	IF NOT bBusy THEN
		fbRun_Color_RTRIG(CLK:=bSetColor, Q=> );
		IF fbRun_Color_RTRIG.Q THEN
			bRunColorWriteCycle:= TRUE;
		END_IF
	
		fbCycleReadTC_TON(IN:= bReadActualTC , PT:=T#1S , Q=> , ET=> );
	
		IF NOT bInitColor AND fActualTcColor = 0 THEN
			bRunColorWriteCycle:=TRUE;
		END_IF

	//Check for correct color in ballast 
	fbColorCheck(IN:= NOT fbColorCheck.Q , PT:= T#2S, Q=> , ET=> );	
	IF fbColorCheck.Q THEN
		IF fColourTemperatureTc <> fActualTcColor  THEN
			bRunColorWriteCycle:=TRUE;			
		END_IF
	END_IF

	
		IF  bRunColorWriteCycle AND NOT GVL_DALI.arrbBlockDTR[nDaliLine] THEN
			bBusy:= TRUE;
			A_ResetRoutine();
			nStep:= 10;
			nErrorID:= 0;
			iStepBeforeError:= 0;	
			GVL_DALI.arrbBlockDTR[nDaliLine] := TRUE;
		END_IF
		
		IF fbCycleReadTC_TON.Q THEN
			bBusy:= TRUE;
			bReadTC:= FALSE;
			A_ResetRoutine();
			nStep:= 100;
			nErrorID:= 0;
			iStepBeforeError:= 0;
		END_IF
	END_IF
	
(* - - - - - - - - - - - - - - - - - - - - - - - - *)
10:(*Set color temperatur to ballast*)
	bStart:= TRUE;
	A_DALICmdSetColourTemperatureTc();
	IF NOT bActionBusy	THEN
		IF bError	THEN
			GVL_DALI.arrbBlockDTR[nDaliLine]:= FALSE;
			nStep:= 0;
		ELSE
			bStart := FALSE;
			nStep:= 11;
		END_IF
	END_IF

11: (* Activate the color temp in ballast*)

	A_DALICmdActivate_DT8();
	
	IF NOT bActionBusy	THEN
		IF bError	THEN
			GVL_DALI.arrbBlockDTR[nDaliLine]:= FALSE;
			nStep:= 0;
		ELSE
			bStart := FALSE;
			nStep:= 100;	
		END_IF
	END_IF	

100: (*Read back current color*)

	A_DALIQueryColourTc();
	IF NOT bActionBusy	THEN
		nStep:= 101;
	END_IF

101: (*Read back color Status*)

	A_DALIQueryColourStatus();
	IF NOT bActionBusy	THEN
		nStep:= 888;
	END_IF
		
888: (*Done step*)
	bBusy:= FALSE;
	nStep:=0;
	nErrorID:= 0;
	iStepBeforeError:= 0;
	bRunColorWriteCycle:= FALSE;
	bInitColor:= TRUE;
	GVL_DALI.arrbBlockDTR[nDaliLine]:= FALSE;
ELSE
	nStep := 0;
END_CASE

//Checking if this FB blocks DT_Telegrams for other ballast

fbDTBlockTimer(IN:=GVL_DALI.arrbBlockDTR[nDaliLine] AND (nStep > 0) AND NOT fbDTBlockTimer.Q , PT:= T#20S , Q=> , ET=> );

IF fbDTBlockTimer.Q THEN
	nStep := 0;
	GVL_DALI.arrbBlockDTR[nDaliLine]:= FALSE;
END_IF

	fActualTcColor := MIREK_TO_KELVIN(fbDALI209QueryColourTc.nColourValue) ;
	nActualColorStatus := fbDALI209QueryColourStatus.nColourStatus;

ACTION A_DALICmdActivate_DT8:
IF eAddressType= E_DALIAddressType.Group THEN
	byAddr		:= byGrpAdr;
	eAddrType	:= E_DALIAddressType.Group;
END_IF

IF eAddressType= E_DALIAddressType.Short THEN
	byAddr		:= byShrtAdr;
	eAddrType	:= E_DALIAddressType.Short;
END_IF

	bActionBusy	:= TRUE;

	fbDALI209Activate(
		bError=> , 
		ipResultMessage=> , 
		bStart:= TRUE, 
		nAddress:= byAddr , 
		eAddressType:= eAddressType, 
		eCommandPriority:=eCommandPriority ,
		bBusy=> );
	

	IF (NOT fbDALI209Activate.bBusy) THEN
		IF fbDALI209Activate.bError THEN
			bError := TRUE;
			nErrorId := fbDALI209Activate.ipResultMessage.nEventId;
		END_IF
		bActionBusy		:= FALSE;
		fbDALI209Activate(bStart:= FALSE);
	END_IF
END_ACTION

ACTION A_DALICmdSetColourTemperatureTc:
IF eAddressType= E_DALIAddressType.Group THEN
	byAddr		:= byGrpAdr;
	eAddrType	:= E_DALIAddressType.Group;
END_IF

IF eAddressType= E_DALIAddressType.Short THEN
	byAddr		:= byShrtAdr;
	eAddrType	:= E_DALIAddressType.Short;
END_IF

	bActionBusy	:= TRUE;

	fbDALI209SetColourTemperatureTc(
		bError=> , 
		ipResultMessage=> , 
		bStart:= TRUE, 
		nAddress:= byAddr , 
		eAddressType:= eAddressType, 
		eCommandPriority:=eCommandPriority , 
		bBusy=> , 
		nColourTemperatureTc:= KELVIN_TO_MIREK(fColourTemperatureTc)
	);
	
	
	
	IF (NOT fbDALI209SetColourTemperatureTc.bBusy) THEN
		IF fbDALI209SetColourTemperatureTc.bError THEN
			bError := TRUE;
			nErrorId := fbDALI209SetColourTemperatureTc.ipResultMessage.nEventId;
		END_IF
		bActionBusy		:= FALSE;
		fbDALI209SetColourTemperatureTc(bStart:= FALSE);
	END_IF
END_ACTION

ACTION A_DALIQueryColourStatus:

	byAddr:= byShrtAdr;

	bActionBusy	:= TRUE;


	fbDALI209QueryColourStatus(
		bError=> , 
		ipResultMessage=> , 
		bStart:= TRUE , 
		nAddress:=byAddr , 
		eAddressType:= Tc3_DALI.E_DALIAddressType.Short, 
		eCommandPriority:= Tc3_DALI.E_DALICommandPriority.Low, 
		bBusy=> , 
		nColourStatus=> );	
	

	IF (NOT fbDALI209QueryColourStatus.bBusy) THEN
		IF fbDALI209QueryColourStatus.bError THEN
			bError := TRUE;
			nErrorId := fbDALI209QueryColourStatus.ipResultMessage.nEventId;
		END_IF
		bActionBusy		:= FALSE;
		fbDALI209QueryColourStatus(bStart:= FALSE);
	END_IF
END_ACTION

ACTION A_DALIQueryColourTc:

	byAddr:= byShrtAdr;

	bActionBusy	:= TRUE;


	fbDALI209QueryColourTc(
		bError=> , 
		ipResultMessage=> , 
		bStart:= TRUE , 
		nAddress:=byAddr , 
		eAddressType:= Tc3_DALI.E_DALIAddressType.Short, 
		eCommandPriority:= Tc3_DALI.E_DALICommandPriority.Low, 
		bBusy=> , 
		eColourValue:= Tc3_DALI.E_DALIColourValue.ColourTemperatureTc , 
		nColourValue=> );	
	

	IF (NOT fbDALI209QueryColourTc.bBusy) THEN
		IF fbDALI209QueryColourTc.bError THEN
			bError := TRUE;
			nErrorId := fbDALI209QueryColourTc.ipResultMessage.nEventId;
		END_IF
		bActionBusy		:= FALSE;
		fbDALI209QueryColourTc(bStart:= FALSE);
	END_IF
END_ACTION

ACTION A_ResetRoutine:

	bError     	:= FALSE;
	nErrorId	:= 0;

	fbDALI209SetColourTemperatureTc (bStart:= FALSE);
	fbDALI209QueryColourStatus(bStart:= FALSE);
	fbDALI209QueryColourTc(bStart:= FALSE);
	fbDALI209Activate(bStart:= FALSE);
END_ACTION

{attribute 'monitoring' := 'call'}
PROPERTY ipDALICommunication : Tc3_DALI.I_DALICommunication
GET
ipDALICommunication := THIS^.ipCommunication;
END_GET
SET
THIS^.ipCommunicationPreset := ipDALICommunication;
END_SET
END_PROPERTY

//| Apply the perset value of IpCommunication if available
//| Return codes:
//|   FALSE: no peset value available
//|   TRUE: has taken the preset value
{attribute 'hide'}
METHOD PRIVATE TrySetCommunication : BOOL
VAR_INPUT
END_VAR
IF ((THIS^.ipCommunication <> THIS^.ipCommunicationPreset) AND (THIS^.ipCommunicationPreset <> 0)) THEN
	THIS^.ipCommunication := THIS^.ipCommunicationPreset;
	THIS^.fbDALI209Activate.ipDALICommunication := THIS^.ipCommunication;
	THIS^.fbDALI209SetColourTemperatureTc.ipDALICommunication := THIS^.ipCommunication;
	THIS^.fbDALI209QueryColourStatus.ipDALICommunication := THIS^.ipCommunication;
	THIS^.fbDALI209QueryColourTc.ipDALICommunication := THIS^.ipCommunication;
	TrySetCommunication := TRUE;
ELSE
	TrySetCommunication := FALSE;
END_IF
END_METHOD

END_FUNCTION_BLOCK

// POUs/DALI/DALI_Devices/BEG/FB_BEG_PD2N_1Pcs
FUNCTION_BLOCK FB_BEG_PD2N_1Pcs
VAR_INPUT
	byShrtAdr					: BYTE;
	bInitialize					: BOOL := TRUE;
	ipCommunication				: I_DALICommunication;
	DALI_LINE_NUM				: INT := 1;	
END_VAR
VAR_OUTPUT
	bInitErr: BOOL;
	bInitDone: BOOL;
END_VAR
VAR
	fbBEGPD2N					: FB_DALI_BEG_PD2N_BMS_V8_FC(0);
	
	fbDelaySetupDALIDevice		: TON;
	tDelayTime					: TIME;
	bInitSensor					: BOOL;
	fbInitDone					: F_TRIG;
	bInitializing				: BOOL;

	bQueryOccupancy				: BOOL;
	bQueryBrightness			: BOOL;

	eEventPriorityOccupancy		: E_DALIEventPriority := E_DALIEVENTPRIORITY.Middle;
	nHoldTimerOccupancy			: WORD := 5; // Value in s. 	
	nReportTimerOccupancy		: BYTE := 120; // Value in s, Preset manufacturer value
	nDeadtimeTimerOccupancy		: WORD := 100; // Value in ms, Predefined Value of DALI Standard
	bCancelHoldTimerOccupancy	: BOOL;
	nSensitivityOccupancy		: BYTE:= 3; //setting Sensivity (0..4) 0 (Off), 1 (Min), 2(Low), 3(High) and 4 (Max)

	bEnableLuxEvent				: BOOL;
	eEventPriorityBrightness	: E_DALIEventPriority := E_DALIEVENTPRIORITY.Middle;
	nDeadtimeTimerBrightness	: WORD := 1500; // Value in ms, Predefined Value of DALI Standard
	nHysteresisBrightness		: BYTE := 2; // Value in %
	nHysteresisMinBrightness	: BYTE := 10; // Absolute Value, depending on the manufacturer specific resolution
	nReportTimerBrightness		: BYTE := 120; // Value in s, Preset manufacturer value

	bAutoRead					: BOOL;
	fbAutoRequestBrightness_TON	: TOF;
	bInitTimeOut: BOOL;
	fbInitTimeOut: Ton;
	nCheckIdx: INT;
	bInitScalesDone: BOOL;
END_VAR
VAR_IN_OUT
	stPirSensorData				: ST_DALI_Sensor;
	arrSensorScales				: ARRAY [1.. 10] OF ST_DALI_SensorScaleMode;
END_VAR

fbBEGPD2N.ipDALICommunication := ipCommunication;

IF NOT bInitScalesDone THEN
	FOR nCheckIdx:= 1 TO 10 DO
		IF arrSensorScales[nCheckIdx].fMeassureMaxSensor = 0 THEN
			arrSensorScales[nCheckIdx].fMeassureMaxSensor := 1;
		END_IF
		IF arrSensorScales[nCheckIdx].fReadMaxSensor = 0 THEN
			arrSensorScales[nCheckIdx].fReadMaxSensor := 1;
		END_IF
	END_FOR
	bInitScalesDone := TRUE;
END_IF

IF ipCommunication <> 0 THEN
	A_BEG_PD2N_1();
END_IF

ACTION A_BEG_PD2N_1:
//Setup parameters
	//Setup Motion part of sensor (Instance 0)
	fbBEGPD2N.bEnableOccupancy := TRUE ;
	fbBEGPD2N.eEventPriorityOccupancy:= eEventPriorityOccupancy;
	fbBEGPD2N.nHoldTimerOccupancy := nHoldTimerOccupancy ;
	fbBEGPD2N.nReportTimerOccupancy := nReportTimerOccupancy;
	fbBEGPD2N.nDeadtimeTimerOccupancy:= nDeadtimeTimerOccupancy;
	fbBEGPD2N.nSensitivityOccupancy:= nSensitivityOccupancy;	
	
	//Setup Brightness part of sensor (Instance 1)
	fbBEGPD2N.bEnableBrightness := bEnableLuxEvent;
	fbBEGPD2N.eEventPriorityBrightness:= eEventPriorityBrightness;
	fbBEGPD2N.nDeadtimeTimerBrightness:= nDeadtimeTimerBrightness;
	fbBEGPD2N.nHysteresisBrightness:= nHysteresisBrightness;
	fbBEGPD2N.nHysteresisMinBrightness:= nHysteresisMinBrightness;
	fbBEGPD2N.nReportTimerBrightness:= nReportTimerBrightness;
	
	
	
//Calculate delay time for init sensor
tDelayTime := INT_TO_TIME((BYTE_TO_INT(byShrtAdr) * 400));	
fbDelaySetupDALIDevice(IN:= bInitialize AND NOT bInitDone , PT:=tDelayTime , Q=> , ET=> );	
	
IF fbDelaySetupDALIDevice.q AND NOT GVL_DALI.arrbBlockDTR[DALI_LINE_NUM] AND NOT bInitErr THEN
	bInitDone := FALSE;
	bInitErr := FALSE;
	bInitSensor:= TRUE;
	GVL_DALI.arrbBlockDTR[DALI_LINE_NUM]:= TRUE;
END_IF

fbAutoRequestBrightness_TON(IN:= NOT fbAutoRequestBrightness_TON.Q  AND NOT stPirSensorData.bQueryBrightness , PT:= (tDelayTime + T#10M) , Q=>bAutoRead , ET=> );

bQueryBrightness:= stPirSensorData.bQueryBrightness OR NOT bAutoRead;

fbBEGPD2N(
	bError=> , 
	ipResultMessage=> , 
	bInitialize:=  bInitSensor, 
	nShortAddress:= byShrtAdr, 
	nOptions:= , 
	bQueryOccupancy:= bQueryOccupancy, 
	bQueryBrightness:= bQueryBrightness, 
	bCancelHoldTimerOccupancy:= bCancelHoldTimerOccupancy, 
	bInitializing=> bInitializing , 
	bReadingOccupancy=> , 
	bReadingBrightness=> , 
	bOccupied=> stPirSensorData.bPrc, 
	nBrightnessLevel=> );


fbInitDone(CLK:=bInitSensor AND bInitializing );	
	IF fbInitDone.Q THEN
		IF NOT bInitTimeOut THEN
			bInitDone := TRUE;
			bInitErr := FALSE;
			GVL_DALI.arrbBlockDTR[DALI_LINE_NUM]:= FALSE;
		ELSE
			bInitErr := TRUE;
			GVL_DALI.arrbBlockDTR[DALI_LINE_NUM]:= FALSE;
		END_IF
	END_IF


fbInitTimeOut(IN:=bInitializing, PT:= T#10S); 

IF fbInitTimeOut.Q THEN
	bInitErr := TRUE;
	GVL_DALI.arrbBlockDTR[DALI_LINE_NUM]:= FALSE;
END_IF

stPirSensorData.bBrightnessRead:= fbBEGPD2N.bReadingBrightness ;

stPirSensorData.fBrightness:= F_fScale(0, arrSensorScales[1].fReadMaxSensor, 0, arrSensorScales[1].fMeassureMaxSensor, 0 , fbBEGPD2N.nBrightnessLevel);
END_ACTION

END_FUNCTION_BLOCK

// POUs/DALI/FUNs/F_fScale
FUNCTION F_fScale : REAL
VAR_INPUT
	fX0, fX1, fY0, fY1, fOffset : REAL;
	nRawValue	:UINT;
END_VAR
VAR
	fDeltaY: REAL;
	fDeltaX: REAL;

END_VAR
VAR_OUTPUT
END_VAR

fDeltaY:= fY1-fY0;
fDeltaX :=fX1-fX0;

IF fDeltaX <=0 THEN
	fDeltaX:=1;
END_IF

F_fScale:= (fDeltaY / fDeltaX) * UINT_TO_REAL(nRawValue) + fOffset;

END_FUNCTION

// POUs/DALI/DALI_Devices/ESYLux/Flat/FB_DALI_ESYLuxFlat_1Pcs
FUNCTION_BLOCK FB_DALI_ESYLuxFlat_1Pcs
VAR_INPUT
	byShrtAdr					: BYTE;
	bInitialize					: BOOL := TRUE;
	ipCommunication				: I_DALICommunication;
	DALI_LINE_NUM				: INT := 1;	
END_VAR
VAR_OUTPUT
END_VAR
VAR
	fbESYLux 					: FB_DALI_Esylux_PD_FLAT_360_BMS(0);
	
	fbDelaySetupDALIDevice		: TON;
	tDelayTime					: TIME;
	bInitSensor					: BOOL;
	fbInitDone					: F_TRIG;

	bQueryOccupancy				: BOOL;
	bQueryBrightness			: BOOL;

	bInitializing				: BOOL;

	eEventPriorityOccupancy		: E_DALIEventPriority := E_DALIEVENTPRIORITY.Middle;
	nHoldTimerOccupancy			: UINT := 5;
	nReportTimerOccupancy		: BYTE := 120; // Value in s, Preset manufacturer value
	nDeadtimeTimerOccupancy		: WORD := 100; // Value in ms, Predefined Value of DALI Standard
	bCancelHoldTimerOccupancy	: BOOL;
	nSensitivityOccupancy		: BYTE := 95; //setting Sensivity 0 = Low 100 = Max
	
	bEnableBrightness			: BOOL := FALSE;
	eEventPriorityBrightness	: E_DALIEventPriority := E_DALIEVENTPRIORITY.MiddleLow;
	nDeadtimeTimerBrightness	: WORD := 1500; // Value in ms, Predefined Value of DALI Standard
	nHysteresisBrightness		: BYTE := 5; // Value in %
	nHysteresisMinBrightness	: BYTE := 40; // Absolute Value, depending on the manufacturer specific resolution
	nReportTimerBrightness		: BYTE := 30; // Value in s, Preset manufacturer value

	bModeLED					: BOOL := FALSE; //LED mode: FALSE: LED disabled, TRUE: LED enabled
	nBrightnessLED				: USINT := 50; //LED brightness (5...100 %).
	
	bAutoRead					: BOOL;
	fbAutoRequestBrightness_TON	: TOF;
	bInitScalesDone				: BOOL;
	nCheckIdx					: INT;
	bInitDone					: BOOL;
	bInitErr					: BOOL;
	bInitTimeOut				: BOOL;
	fbInitTimeOut				: TON;
END_VAR
VAR_IN_OUT
	stPirSensorData				: ST_DALI_Sensor;
	arrSensorScales				: ARRAY [1.. 10] OF ST_DALI_SensorScaleMode;
END_VAR

fbESYLux.ipDALICommunication:= ipCommunication;

IF NOT bInitScalesDone THEN
	FOR nCheckIdx:= 1 TO 10 DO
		IF arrSensorScales[nCheckIdx].fMeassureMaxSensor = 0 THEN
			arrSensorScales[nCheckIdx].fMeassureMaxSensor := 1;
		END_IF
		IF arrSensorScales[nCheckIdx].fReadMaxSensor = 0 THEN
			arrSensorScales[nCheckIdx].fReadMaxSensor := 1;
		END_IF
	END_FOR
	bInitScalesDone := TRUE;
END_IF

IF ipCommunication <> 0 THEN
	A_ESYLux_1();
END_IF

ACTION A_ESYLux_1:
//Setup parameters
	//Setup Motion part of sensor (Instance 1)

	fbESYLux.bEnableOccupancy := TRUE;
	fbESYLux.eEventPriorityOccupancy:= eEventPriorityOccupancy;
	fbESYLux.nHoldTimerOccupancy := nHoldTimerOccupancy ;
	fbESYLux.nReportTimerOccupancy := nReportTimerOccupancy;
	fbESYLux.nDeadtimeTimerOccupancy:= nDeadtimeTimerOccupancy;
	fbESYLux.nSensitivityOccupancy:= nSensitivityOccupancy;
	
	
	//Setup Brightness part of sensor (Instance 2)
	fbESYLux.bEnableBrightness:= bEnableBrightness;
	fbESYLux.eEventPriorityBrightness:= eEventPriorityBrightness;
	fbESYLux.nDeadtimeTimerBrightness:= nDeadtimeTimerBrightness;
	fbESYLux.nHysteresisBrightness:= nHysteresisBrightness;
	fbESYLux.nHysteresisMinBrightness:= nHysteresisMinBrightness;
	fbESYLux.nReportTimerBrightness:= nReportTimerBrightness;

	fbESYLux.bModeLED:= bModeLED;
	fbESYLux.nBrightnessLED:= nBrightnessLED;
	
	
//Calculate delay time for init sensor
tDelayTime := INT_TO_TIME((BYTE_TO_INT(byShrtAdr) * 400));	
fbDelaySetupDALIDevice(IN:= bInitialize AND NOT bInitDone , PT:=tDelayTime , Q=> , ET=> );	
	
IF fbDelaySetupDALIDevice.q AND NOT GVL_DALI.arrbBlockDTR[DALI_LINE_NUM] AND NOT bInitErr THEN
	bInitDone := FALSE;
	bInitErr := FALSE;
	bInitSensor:= TRUE;
	GVL_DALI.arrbBlockDTR[DALI_LINE_NUM]:= TRUE;
END_IF

fbAutoRequestBrightness_TON(IN:= NOT fbAutoRequestBrightness_TON.Q  AND NOT stPirSensorData.bQueryBrightness , PT:= (tDelayTime + T#12M) , Q=>bAutoRead , ET=> );

bQueryBrightness:= stPirSensorData.bQueryBrightness OR NOT bAutoRead;

fbESYLux(
	bInitialize:= bInitSensor, 
	nShortAddress:= byShrtAdr, 
	nOptions:= , 
	bQueryPushButton:= , 
	bQueryOccupancy:= bQueryOccupancy, 
	bQueryBrightness:= bQueryBrightness, 
	bCancelHoldTimerOccupancy:= bCancelHoldTimerOccupancy, 
	bInitializing=> bInitializing , 
	bReadingPushButton=> , 
	bReadingOccupancy=> , 
	bReadingBrightness=> , 
	nPushButtonEvent=> , 
	bOccupied=> stPirSensorData.bPrc, 
	nBrightnessLevel=> );

fbInitDone(CLK:=bInitSensor AND bInitializing );	
	IF fbInitDone.Q THEN
		IF NOT bInitTimeOut THEN
			bInitDone := TRUE;
			bInitErr := FALSE;
			GVL_DALI.arrbBlockDTR[DALI_LINE_NUM]:= FALSE;
		ELSE
			bInitErr := TRUE;
			GVL_DALI.arrbBlockDTR[DALI_LINE_NUM]:= FALSE;
		END_IF
	END_IF


fbInitTimeOut(IN:=bInitializing, PT:= T#10S); 

IF fbInitTimeOut.Q THEN
	bInitErr := TRUE;
	GVL_DALI.arrbBlockDTR[DALI_LINE_NUM]:= FALSE;
END_IF

stPirSensorData.bBrightnessRead:= fbESYLux.bReadingBrightness ;

stPirSensorData.fBrightness:= F_fScale(0, arrSensorScales[1].fReadMaxSensor, 0, arrSensorScales[1].fMeassureMaxSensor, 0 , fbESYLux.nBrightnessLevel);
END_ACTION

END_FUNCTION_BLOCK

// POUs/DALI/DALI_Devices/ESYLux/FB_DALI_ESYLux_1Pcs
FUNCTION_BLOCK FB_DALI_ESYLux_1Pcs
VAR_INPUT
	byShrtAdr					: BYTE;
	bInitialize					: BOOL := TRUE;
	ipCommunication				: I_DALICommunication;
	DALI_LINE_NUM				: INT := 1;	
END_VAR
VAR_OUTPUT
END_VAR
VAR
	fbESYLux 					: FB_DALI_Esylux_PD_C_360_BMS(0);
	
	fbDelaySetupDALIDevice		: TON;
	tDelayTime					: TIME;
	bInitSensor					: BOOL;
	fbInitDone					: F_TRIG;

	bQueryOccupancy				: BOOL;
	bQueryBrightness			: BOOL;

	bInitializing				: BOOL;

	eEventPriorityOccupancy		: E_DALIEventPriority := E_DALIEVENTPRIORITY.Middle;
	nHoldTimerOccupancy			: UINT := 5;
	nReportTimerOccupancy		: BYTE := 120; // Value in s, Preset manufacturer value
	nDeadtimeTimerOccupancy		: WORD := 100; // Value in ms, Predefined Value of DALI Standard
	bCancelHoldTimerOccupancy	: BOOL;
	nSensitivityOccupancy		: BYTE := 95; //setting Sensivity 0 = Low 100 = Max
	
	bEnableBrightness			: BOOL := FALSE;
	eEventPriorityBrightness	: E_DALIEventPriority := E_DALIEVENTPRIORITY.MiddleLow;
	nDeadtimeTimerBrightness	: WORD := 1500; // Value in ms, Predefined Value of DALI Standard
	nHysteresisBrightness		: BYTE := 5; // Value in %
	nHysteresisMinBrightness	: BYTE := 40; // Absolute Value, depending on the manufacturer specific resolution
	nReportTimerBrightness		: BYTE := 30; // Value in s, Preset manufacturer value

	bModeLED					: BOOL := FALSE; //LED mode: FALSE: LED disabled, TRUE: LED enabled
	nBrightnessLED				: USINT := 50; //LED brightness (5...100 %).
	
	bAutoRead					: BOOL;
	fbAutoRequestBrightness_TON	: TOF;
	bInitScalesDone				: BOOL;
	nCheckIdx					: INT;
	bInitDone					: BOOL;
	bInitErr					: BOOL;
	bInitTimeOut				: BOOL;
	fbInitTimeOut				: TON;
END_VAR
VAR_IN_OUT
	stPirSensorData				: ST_DALI_Sensor;
	arrSensorScales				: ARRAY [1.. 10] OF ST_DALI_SensorScaleMode;
END_VAR

fbESYLux.ipDALICommunication:= ipCommunication;

IF NOT bInitScalesDone THEN
	FOR nCheckIdx:= 1 TO 10 DO
		IF arrSensorScales[nCheckIdx].fMeassureMaxSensor = 0 THEN
			arrSensorScales[nCheckIdx].fMeassureMaxSensor := 1;
		END_IF
		IF arrSensorScales[nCheckIdx].fReadMaxSensor = 0 THEN
			arrSensorScales[nCheckIdx].fReadMaxSensor := 1;
		END_IF
	END_FOR
	bInitScalesDone := TRUE;
END_IF

IF ipCommunication <> 0 THEN
	A_ESYLux_1();
END_IF

ACTION A_ESYLux_1:
//Setup parameters
	//Setup Motion part of sensor (Instance 0)

	fbESYLux.bEnableOccupancy := TRUE;
	fbESYLux.eEventPriorityOccupancy:= eEventPriorityOccupancy;
	fbESYLux.nHoldTimerOccupancy := nHoldTimerOccupancy ;
	fbESYLux.nReportTimerOccupancy := nReportTimerOccupancy;
	fbESYLux.nDeadtimeTimerOccupancy:= nDeadtimeTimerOccupancy;
	fbESYLux.nSensitivityOccupancy:= nSensitivityOccupancy;
	
	
	//Setup Brightness part of sensor (Instance 1)
	fbESYLux.bEnableBrightness:= bEnableBrightness;
	fbESYLux.eEventPriorityBrightness:= eEventPriorityBrightness;
	fbESYLux.nDeadtimeTimerBrightness:= nDeadtimeTimerBrightness;
	fbESYLux.nHysteresisBrightness:= nHysteresisBrightness;
	fbESYLux.nHysteresisMinBrightness:= nHysteresisMinBrightness;
	fbESYLux.nReportTimerBrightness:= nReportTimerBrightness;

	fbESYLux.bModeLED:= bModeLED;
	fbESYLux.nBrightnessLED:= nBrightnessLED;
	
	
//Calculate delay time for init sensor
tDelayTime := INT_TO_TIME((BYTE_TO_INT(byShrtAdr) * 400));	
fbDelaySetupDALIDevice(IN:= bInitialize AND NOT bInitDone , PT:=tDelayTime , Q=> , ET=> );	
	
IF fbDelaySetupDALIDevice.q AND NOT GVL_DALI.arrbBlockDTR[DALI_LINE_NUM] AND NOT bInitErr THEN
	bInitDone := FALSE;
	bInitErr := FALSE;
	bInitSensor:= TRUE;
	GVL_DALI.arrbBlockDTR[DALI_LINE_NUM]:= TRUE;
END_IF

fbAutoRequestBrightness_TON(IN:= NOT fbAutoRequestBrightness_TON.Q  AND NOT stPirSensorData.bQueryBrightness , PT:= (tDelayTime + T#12M) , Q=>bAutoRead , ET=> );

bQueryBrightness:= stPirSensorData.bQueryBrightness OR NOT bAutoRead;

fbESYLux(
	bInitialize:= bInitSensor, 
	nShortAddress:= byShrtAdr, 
	nOptions:= , 
	bQueryPushButton1:= , 
	bQueryPushButton2:= , 
	bQueryOccupancy:= bQueryOccupancy, 
	bQueryBrightness:= bQueryBrightness, 
	bCancelHoldTimerOccupancy:= bCancelHoldTimerOccupancy, 
	bInitializing=> bInitializing , 
	bReadingPushButton1=> , 
	bReadingPushButton2=> , 
	bReadingOccupancy=> , 
	bReadingBrightness=> , 
	nPushButton1Event=> , 
	nPushButton2Event=> , 
	bOccupied=> stPirSensorData.bPrc, 
	nBrightnessLevel=> );


fbInitDone(CLK:=bInitSensor AND bInitializing );	
	IF fbInitDone.Q THEN
		IF NOT bInitTimeOut THEN
			bInitDone := TRUE;
			bInitErr := FALSE;
			GVL_DALI.arrbBlockDTR[DALI_LINE_NUM]:= FALSE;
		ELSE
			bInitErr := TRUE;
			GVL_DALI.arrbBlockDTR[DALI_LINE_NUM]:= FALSE;
		END_IF
	END_IF


fbInitTimeOut(IN:=bInitializing, PT:= T#10S); 

IF fbInitTimeOut.Q THEN
	bInitErr := TRUE;
	GVL_DALI.arrbBlockDTR[DALI_LINE_NUM]:= FALSE;
END_IF

stPirSensorData.bBrightnessRead:= fbESYLux.bReadingBrightness ;

stPirSensorData.fBrightness:= F_fScale(0, arrSensorScales[1].fReadMaxSensor, 0, arrSensorScales[1].fMeassureMaxSensor, 0 , fbESYLux.nBrightnessLevel);
END_ACTION

END_FUNCTION_BLOCK

// POUs/DALI/DALI_Devices/ESYLux/FB_DALI_ESYLux_2Pcs
FUNCTION_BLOCK FB_DALI_ESYLux_2Pcs
VAR_INPUT
	byShrtAdr					: BYTE;
	bInitialize					: BOOL := TRUE;
	ipCommunication				: I_DALICommunication;
	DALI_LINE_NUM				: INT := 1;	
END_VAR
VAR_OUTPUT
	arrInitErr: ARRAY [1.. nNumberOfSensors] OF BOOL;
	arrInitDone: ARRAY [1.. nNumberOfSensors] OF BOOL;
END_VAR
VAR
	arrEsylux_PD_C				: ARRAY [1.. nNumberOfSensors] OF FB_DALI_Esylux_PD_C_360_BMS(0);
	
	arrDelaySetupDALIDevice		: ARRAY [1.. nNumberOfSensors] Of TON;
	arrtDelayTime				: ARRAY [1.. nNumberOfSensors] OF TIME;
	arrInitSensor				: ARRAY [1.. nNumberOfSensors] OF BOOL;
	arrInitDone_FTrig			: ARRAY [1.. nNumberOfSensors] OF F_TRIG;
	arrInitializing				: ARRAY [1.. nNumberOfSensors] OF BOOL;

	bQueryBrightness 			: BOOL;
	bQueryOccupancy				: BOOL;

	eEventPriorityOccupancy		: E_DALIEventPriority := E_DALIEVENTPRIORITY.Middle;
	nHoldTimerOccupancy			: UINT := 5;
	nReportTimerOccupancy		: BYTE := 120; // Value in s, Preset manufacturer value
	nDeadtimeTimerOccupancy		: WORD := 100; // Value in ms, Predefined Value of DALI Standard
	bCancelHoldTimerOccupancy	: BOOL;
	nSensitivityOccupancy		: BYTE := 95; //setting Sensivity 0 = Low 100 = Max
	
	bEnableBrightness			: BOOL := FALSE;
	eEventPriorityBrightness	: E_DALIEventPriority := E_DALIEVENTPRIORITY.MiddleLow;
	nDeadtimeTimerBrightness	: WORD := 1500; // Value in ms, Predefined Value of DALI Standard
	nHysteresisBrightness		: BYTE := 5; // Value in %
	nHysteresisMinBrightness	: BYTE := 40; // Absolute Value, depending on the manufacturer specific resolution
	nReportTimerBrightness		: BYTE := 30; // Value in s, Preset manufacturer value

	bModeLED					: BOOL := FALSE; //LED mode: FALSE: LED disabled, TRUE: LED enabled
	nBrightnessLED				: USINT := 50; //LED brightness (5...100 %).

	bAutoRead					: BOOL;
	fbAutoRequestBrightness_TON	: TOF;
	bInitTimeOut				: BOOL;
	fbInitTimeOut				: ARRAY [1.. nNumberOfSensors] OF TON;
	nIdxScan					: BYTE;
	nPirIdxOn					: BYTE;
	nBrightnessIdx				: BYTE;
	fBrightness_1				: REAL;
	fBrightness_2				: REAL;
	fBrightness_3				: REAL;
	bInitDone					: BOOL;
	bInitScalesDone				: BOOL;
	
	nCheckIdx: INT;
END_VAR
VAR_IN_OUT
	stPirSensorData				: ST_DALI_Sensor;
	arrSensorScales				: ARRAY [1.. 10] OF ST_DALI_SensorScaleMode;
END_VAR

VAR CONSTANT
	nNumberOfSensors: BYTE := 2;
END_VAR

arrEsylux_PD_C[1].ipDALICommunication := ipCommunication;
arrEsylux_PD_C[2].ipDALICommunication := ipCommunication;


IF NOT bInitScalesDone THEN
	FOR nCheckIdx:= 1 TO 10 DO
		IF arrSensorScales[nCheckIdx].fMeassureMaxSensor = 0 THEN
			arrSensorScales[nCheckIdx].fMeassureMaxSensor := 1;
		END_IF
		IF arrSensorScales[nCheckIdx].fReadMaxSensor = 0 THEN
			arrSensorScales[nCheckIdx].fReadMaxSensor := 1;
		END_IF
	END_FOR
	bInitScalesDone := TRUE;
END_IF

IF ipCommunication <> 0 THEN
	A_ESYLux_2Pcs();
END_IF

ACTION A_ESYLux_2Pcs:


FOR nIdxScan := 1 TO nNumberOfSensors DO
	//Setup parameters
	//Setup Motion part of sensor (Instance 0)
	arrEsylux_PD_C[nIdxScan].bEnableOccupancy := TRUE;
	arrEsylux_PD_C[nIdxScan].eEventPriorityOccupancy:= eEventPriorityOccupancy;
	arrEsylux_PD_C[nIdxScan].nHoldTimerOccupancy := nHoldTimerOccupancy ;
	arrEsylux_PD_C[nIdxScan].nDeadtimeTimerOccupancy:= 	nDeadtimeTimerOccupancy;
	arrEsylux_PD_C[nIdxScan].nReportTimerOccupancy:= nReportTimerOccupancy;
	arrEsylux_PD_C[nIdxScan].nSensitivityOccupancy:= 100;
	
	//Setup Brightness part of sensor (Instance 1)
	arrEsylux_PD_C[nIdxScan].bEnableBrightness:= bEnableBrightness;
	arrEsylux_PD_C[nIdxScan].eEventPriorityBrightness:= eEventPriorityBrightness;
	arrEsylux_PD_C[nIdxScan].nDeadtimeTimerBrightness:= nDeadtimeTimerBrightness;
	arrEsylux_PD_C[nIdxScan].nHysteresisBrightness:= nHysteresisBrightness;
	arrEsylux_PD_C[nIdxScan].nHysteresisMinBrightness:= nHysteresisMinBrightness;
	arrEsylux_PD_C[nIdxScan].nReportTimerBrightness:= nReportTimerBrightness;

	arrEsylux_PD_C[nIdxScan].bModeLED:= bModeLED;
	arrEsylux_PD_C[nIdxScan].nBrightnessLED:= nBrightnessLED;
	
		
		
	//Calculate delay time for init sensor
	arrtDelayTime[nIdxScan] := INT_TO_TIME((BYTE_TO_INT((byShrtAdr + nIdxScan)-1) * 400));	
	arrDelaySetupDALIDevice[nIdxScan](IN:= bInitialize , PT:=arrtDelayTime[nIdxScan] , Q=> , ET=> );	
		
	IF arrDelaySetupDALIDevice[nIdxScan].q AND NOT GVL_DALI.arrbBlockDTR[DALI_LINE_NUM] AND NOT (arrInitDone[nIdxScan] OR arrInitErr[nIdxScan]) THEN
		arrInitSensor[nIdxScan]:= TRUE;
		GVL_DALI.arrbBlockDTR[DALI_LINE_NUM]:= TRUE;
	END_IF
	
	bQueryBrightness:= stPirSensorData.bQueryBrightness OR NOT bAutoRead;
	
	fbAutoRequestBrightness_TON(IN:= NOT fbAutoRequestBrightness_TON.Q  AND NOT stPirSensorData.bQueryBrightness , PT:= (arrtDelayTime[nIdxScan] + T#12M) , Q=>bAutoRead , ET=> );
	
	bQueryOccupancy:= NOT bAutoRead OR stPirSensorData.bQueryBrightness;
	
	arrEsylux_PD_C[nIdxScan](
		bError=> , 
		ipResultMessage=> , 
		bInitialize:=  arrInitSensor[nIdxScan], 
		nShortAddress:= (byShrtAdr + nIdxScan)-1 , 
		nOptions:= , 
		bQueryOccupancy:= bQueryOccupancy, 
		bQueryBrightness:= bQueryBrightness, 
		bCancelHoldTimerOccupancy:= bCancelHoldTimerOccupancy, 
		bInitializing=> arrInitializing[nIdxScan] , 
		bReadingOccupancy=> , 
		bReadingBrightness=> , 
		bOccupied=> , 
		nBrightnessLevel=> );
	
	arrInitDone_FTrig[nIdxScan](CLK:=arrInitializing[nIdxScan] );	
		IF arrInitDone_FTrig[nIdxScan].Q THEN
			IF NOT bInitTimeOut THEN
				arrInitDone[nIdxScan] := TRUE;
				GVL_DALI.arrbBlockDTR[DALI_LINE_NUM]:= FALSE;
			ELSE
				arrInitErr[nIdxScan] := TRUE;
				GVL_DALI.arrbBlockDTR[DALI_LINE_NUM]:= FALSE;
			END_IF
		END_IF
		
	fbInitTimeOut[nIdxScan](IN:=arrInitSensor[nIdxScan] AND NOT arrInitDone[nIdxScan], PT:= T#10S); 
	
	IF fbInitTimeOut[nIdxScan].Q THEN
		arrInitErr[nIdxScan] := TRUE;
		GVL_DALI.arrbBlockDTR[DALI_LINE_NUM]:= FALSE;
	END_IF
END_FOR

stPirSensorData.bPrc:= FALSE;
FOR nPirIdxOn:= 1 TO nNumberOfSensors DO
	IF arrEsylux_PD_C[nPirIdxOn].bOccupied THEN
		stPirSensorData.bPrc:= TRUE;
		EXIT;
	END_IF
END_FOR

stPirSensorData.bBrightnessRead:= arrEsylux_PD_C[1].bReadingBrightness OR arrEsylux_PD_C[2].bReadingBrightness ;


fBrightness_1:= F_fScale(0, arrSensorScales[1].fReadMaxSensor, 0, arrSensorScales[1].fMeassureMaxSensor, 0, arrEsylux_PD_C[1].nBrightnessLevel);
fBrightness_2:= F_fScale(0, arrSensorScales[2].fReadMaxSensor, 0, arrSensorScales[2].fMeassureMaxSensor, 0, arrEsylux_PD_C[2].nBrightnessLevel);


IF fBrightness_1 <> 0 THEN
	stPirSensorData.fBrightness:= fBrightness_1;
END_IF
IF fBrightness_2 <> 0 THEN
	stPirSensorData.fBrightness:= MIN(fBrightness_2, stPirSensorData.fBrightness);
END_IF

IF NOT bInitialize THEN
	FOR nIdxScan := 1 TO nNumberOfSensors DO
		arrInitSensor[nIdxScan]:= FALSE;
		fbInitTimeOut[nIdxScan](IN:= FALSE);
		arrInitDone[nIdxScan] := FALSE;
		arrInitErr[nIdxScan] := FALSE;
	END_FOR
END_IF
END_ACTION

END_FUNCTION_BLOCK

// POUs/DALI/DALI_Devices/ESYLux/FB_DALI_ESYLux_3Pcs
FUNCTION_BLOCK FB_DALI_ESYLux_3Pcs
VAR_INPUT
	byShrtAdr					: BYTE;
	bInitialize					: BOOL := TRUE;
	ipCommunication				: I_DALICommunication;
	DALI_LINE_NUM				: INT := 1;	
END_VAR
VAR_OUTPUT
	arrInitErr: ARRAY [1.. nNumberOfSensors] OF BOOL;
	arrInitDone: ARRAY [1.. nNumberOfSensors] OF BOOL;
END_VAR
VAR
	arrEsylux_PD_C				: ARRAY [1.. nNumberOfSensors] OF FB_DALI_Esylux_PD_C_360_BMS(0);
	
	arrDelaySetupDALIDevice		: ARRAY [1.. nNumberOfSensors] Of TON;
	arrtDelayTime				: ARRAY [1.. nNumberOfSensors] OF TIME;
	arrInitSensor				: ARRAY [1.. nNumberOfSensors] OF BOOL;
	arrInitDone_FTrig			: ARRAY [1.. nNumberOfSensors] OF F_TRIG;
	arrInitializing				: ARRAY [1.. nNumberOfSensors] OF BOOL;

	bQueryBrightness 			: BOOL;
	bQueryOccupancy				: BOOL;

	eEventPriorityOccupancy		: E_DALIEventPriority := E_DALIEVENTPRIORITY.Middle;
	nHoldTimerOccupancy			: UINT := 5;
	nReportTimerOccupancy		: BYTE := 120; // Value in s, Preset manufacturer value
	nDeadtimeTimerOccupancy		: WORD := 100; // Value in ms, Predefined Value of DALI Standard
	bCancelHoldTimerOccupancy	: BOOL;
	nSensitivityOccupancy		: BYTE := 95; //setting Sensivity 0 = Low 100 = Max
	
	bEnableBrightness			: BOOL := FALSE;
	eEventPriorityBrightness	: E_DALIEventPriority := E_DALIEVENTPRIORITY.MiddleLow;
	nDeadtimeTimerBrightness	: WORD := 1500; // Value in ms, Predefined Value of DALI Standard
	nHysteresisBrightness		: BYTE := 5; // Value in %
	nHysteresisMinBrightness	: BYTE := 40; // Absolute Value, depending on the manufacturer specific resolution
	nReportTimerBrightness		: BYTE := 30; // Value in s, Preset manufacturer value

	bModeLED					: BOOL := FALSE; //LED mode: FALSE: LED disabled, TRUE: LED enabled
	nBrightnessLED				: USINT := 50; //LED brightness (5...100 %).

	bAutoRead					: BOOL;
	fbAutoRequestBrightness_TON	: TOF;
	bInitTimeOut				: BOOL;
	fbInitTimeOut				: ARRAY [1.. nNumberOfSensors] OF TON;
	nIdxScan					: BYTE;
	nPirIdxOn					: BYTE;
	nBrightnessIdx				: BYTE;
	fBrightness_1				: REAL;
	fBrightness_2				: REAL;
	fBrightness_3				: REAL;
	bInitDone					: BOOL;
	bInitScalesDone				: BOOL;
	
	nCheckIdx: INT;
END_VAR
VAR_IN_OUT
	stPirSensorData				: ST_DALI_Sensor;
	arrSensorScales				: ARRAY [1.. 10] OF ST_DALI_SensorScaleMode;
END_VAR

VAR CONSTANT
	nNumberOfSensors: BYTE := 3;
END_VAR

arrEsylux_PD_C[1].ipDALICommunication := ipCommunication;
arrEsylux_PD_C[2].ipDALICommunication := ipCommunication;
arrEsylux_PD_C[3].ipDALICommunication := ipCommunication;

IF NOT bInitScalesDone THEN
	FOR nCheckIdx:= 1 TO 10 DO
		IF arrSensorScales[nCheckIdx].fMeassureMaxSensor = 0 THEN
			arrSensorScales[nCheckIdx].fMeassureMaxSensor := 1;
		END_IF
		IF arrSensorScales[nCheckIdx].fReadMaxSensor = 0 THEN
			arrSensorScales[nCheckIdx].fReadMaxSensor := 1;
		END_IF
	END_FOR
	bInitScalesDone := TRUE;
END_IF

IF ipCommunication <> 0 THEN
	A_ESYLux_3Pcs();
END_IF

ACTION A_ESYLux_3Pcs:


FOR nIdxScan := 1 TO nNumberOfSensors DO
	//Setup parameters
	//Setup Motion part of sensor (Instance 0)
	arrEsylux_PD_C[nIdxScan].bEnableOccupancy := TRUE;
	arrEsylux_PD_C[nIdxScan].eEventPriorityOccupancy:= eEventPriorityOccupancy;
	arrEsylux_PD_C[nIdxScan].nHoldTimerOccupancy := nHoldTimerOccupancy ;
	arrEsylux_PD_C[nIdxScan].nDeadtimeTimerOccupancy:= 	nDeadtimeTimerOccupancy;
	arrEsylux_PD_C[nIdxScan].nReportTimerOccupancy:= nReportTimerOccupancy;
	arrEsylux_PD_C[nIdxScan].nSensitivityOccupancy:= 100;
	
	//Setup Brightness part of sensor (Instance 1)
	arrEsylux_PD_C[nIdxScan].bEnableBrightness:= bEnableBrightness;
	arrEsylux_PD_C[nIdxScan].eEventPriorityBrightness:= eEventPriorityBrightness;
	arrEsylux_PD_C[nIdxScan].nDeadtimeTimerBrightness:= nDeadtimeTimerBrightness;
	arrEsylux_PD_C[nIdxScan].nHysteresisBrightness:= nHysteresisBrightness;
	arrEsylux_PD_C[nIdxScan].nHysteresisMinBrightness:= nHysteresisMinBrightness;
	arrEsylux_PD_C[nIdxScan].nReportTimerBrightness:= nReportTimerBrightness;

	arrEsylux_PD_C[nIdxScan].bModeLED:= bModeLED;
	arrEsylux_PD_C[nIdxScan].nBrightnessLED:= nBrightnessLED;
	
		
		
	//Calculate delay time for init sensor
	arrtDelayTime[nIdxScan] := INT_TO_TIME((BYTE_TO_INT((byShrtAdr + nIdxScan)-1) * 400));	
	arrDelaySetupDALIDevice[nIdxScan](IN:= bInitialize , PT:=arrtDelayTime[nIdxScan] , Q=> , ET=> );	
		
	IF arrDelaySetupDALIDevice[nIdxScan].q AND NOT GVL_DALI.arrbBlockDTR[DALI_LINE_NUM] AND NOT (arrInitDone[nIdxScan] OR arrInitErr[nIdxScan]) THEN
		arrInitSensor[nIdxScan]:= TRUE;
		GVL_DALI.arrbBlockDTR[DALI_LINE_NUM]:= TRUE;
	END_IF
	
	bQueryBrightness:= stPirSensorData.bQueryBrightness OR NOT bAutoRead;
	
	fbAutoRequestBrightness_TON(IN:= NOT fbAutoRequestBrightness_TON.Q  AND NOT stPirSensorData.bQueryBrightness , PT:= (arrtDelayTime[nIdxScan] + T#12M) , Q=>bAutoRead , ET=> );
	
	bQueryOccupancy:= NOT bAutoRead OR stPirSensorData.bQueryBrightness;
	
	arrEsylux_PD_C[nIdxScan](
		bError=> , 
		ipResultMessage=> , 
		bInitialize:=  arrInitSensor[nIdxScan], 
		nShortAddress:= (byShrtAdr + nIdxScan)-1 , 
		nOptions:= , 
		bQueryOccupancy:= bQueryOccupancy, 
		bQueryBrightness:= bQueryBrightness, 
		bCancelHoldTimerOccupancy:= bCancelHoldTimerOccupancy, 
		bInitializing=> arrInitializing[nIdxScan] , 
		bReadingOccupancy=> , 
		bReadingBrightness=> , 
		bOccupied=> , 
		nBrightnessLevel=> );
	
	arrInitDone_FTrig[nIdxScan](CLK:=arrInitializing[nIdxScan] );	
		IF arrInitDone_FTrig[nIdxScan].Q THEN
			IF NOT bInitTimeOut THEN
				arrInitDone[nIdxScan] := TRUE;
				GVL_DALI.arrbBlockDTR[DALI_LINE_NUM]:= FALSE;
			ELSE
				arrInitErr[nIdxScan] := TRUE;
				GVL_DALI.arrbBlockDTR[DALI_LINE_NUM]:= FALSE;
			END_IF
		END_IF
		
	fbInitTimeOut[nIdxScan](IN:=arrInitSensor[nIdxScan] AND NOT arrInitDone[nIdxScan], PT:= T#10S); 
	
	IF fbInitTimeOut[nIdxScan].Q THEN
		arrInitErr[nIdxScan] := TRUE;
		GVL_DALI.arrbBlockDTR[DALI_LINE_NUM]:= FALSE;
	END_IF
END_FOR

stPirSensorData.bPrc:= FALSE;
FOR nPirIdxOn:= 1 TO nNumberOfSensors DO
	IF arrEsylux_PD_C[nPirIdxOn].bOccupied THEN
		stPirSensorData.bPrc:= TRUE;
		EXIT;
	END_IF
END_FOR

stPirSensorData.bBrightnessRead:= arrEsylux_PD_C[1].bReadingBrightness OR arrEsylux_PD_C[2].bReadingBrightness OR arrEsylux_PD_C[3].bReadingBrightness;

fBrightness_1:= F_fScale(0, arrSensorScales[1].fReadMaxSensor, 0, arrSensorScales[1].fMeassureMaxSensor, 0, arrEsylux_PD_C[1].nBrightnessLevel);
fBrightness_2:= F_fScale(0, arrSensorScales[2].fReadMaxSensor, 0, arrSensorScales[2].fMeassureMaxSensor, 0, arrEsylux_PD_C[2].nBrightnessLevel);
fBrightness_3:= F_fScale(0, arrSensorScales[3].fReadMaxSensor, 0, arrSensorScales[3].fMeassureMaxSensor, 0, arrEsylux_PD_C[3].nBrightnessLevel);


IF fBrightness_1 <> 0 THEN
	stPirSensorData.fBrightness:= fBrightness_1;
END_IF
IF fBrightness_2 <> 0 THEN
	stPirSensorData.fBrightness:= MIN(fBrightness_2, stPirSensorData.fBrightness);
END_IF
IF fBrightness_3 <> 0 THEN
	stPirSensorData.fBrightness:=  MIN(fBrightness_3, stPirSensorData.fBrightness);
END_IF

IF NOT bInitialize THEN
	FOR nIdxScan := 1 TO nNumberOfSensors DO
		arrInitSensor[nIdxScan]:= FALSE;
		fbInitTimeOut[nIdxScan](IN:= FALSE);
		arrInitDone[nIdxScan] := FALSE;
		arrInitErr[nIdxScan] := FALSE;
	END_FOR
END_IF
END_ACTION

END_FUNCTION_BLOCK

// POUs/DALI/DALI_Devices/ESYLux/FB_DALI_ESYLux_4Pcs
FUNCTION_BLOCK FB_DALI_ESYLux_4Pcs
VAR_INPUT
	byShrtAdr					: BYTE;
	bInitialize					: BOOL := TRUE;
	ipCommunication				: I_DALICommunication;
	DALI_LINE_NUM				: INT := 1;	
END_VAR
VAR_OUTPUT
	arrInitErr: ARRAY [1.. nNumberOfSensors] OF BOOL;
	arrInitDone: ARRAY [1.. nNumberOfSensors] OF BOOL;
END_VAR
VAR
	arrEsylux_PD_C				: ARRAY [1.. nNumberOfSensors] OF FB_DALI_Esylux_PD_C_360_BMS(0);
	
	arrDelaySetupDALIDevice		: ARRAY [1.. nNumberOfSensors] Of TON;
	arrtDelayTime				: ARRAY [1.. nNumberOfSensors] OF TIME;
	arrInitSensor				: ARRAY [1.. nNumberOfSensors] OF BOOL;
	arrInitDone_FTrig			: ARRAY [1.. nNumberOfSensors] OF F_TRIG;
	arrInitializing				: ARRAY [1.. nNumberOfSensors] OF BOOL;

	bQueryBrightness 			: BOOL;
	bQueryOccupancy				: BOOL;

	eEventPriorityOccupancy		: E_DALIEventPriority := E_DALIEVENTPRIORITY.Middle;
	nHoldTimerOccupancy			: UINT := 5;
	nReportTimerOccupancy		: BYTE := 120; // Value in s, Preset manufacturer value
	nDeadtimeTimerOccupancy		: WORD := 100; // Value in ms, Predefined Value of DALI Standard
	bCancelHoldTimerOccupancy	: BOOL;
	nSensitivityOccupancy		: BYTE := 95; //setting Sensivity 0 = Low 100 = Max
	
	bEnableBrightness			: BOOL := FALSE;
	eEventPriorityBrightness	: E_DALIEventPriority := E_DALIEVENTPRIORITY.MiddleLow;
	nDeadtimeTimerBrightness	: WORD := 1500; // Value in ms, Predefined Value of DALI Standard
	nHysteresisBrightness		: BYTE := 5; // Value in %
	nHysteresisMinBrightness	: BYTE := 40; // Absolute Value, depending on the manufacturer specific resolution
	nReportTimerBrightness		: BYTE := 30; // Value in s, Preset manufacturer value

	bModeLED					: BOOL := FALSE; //LED mode: FALSE: LED disabled, TRUE: LED enabled
	nBrightnessLED				: USINT := 50; //LED brightness (5...100 %).

	bAutoRead					: BOOL;
	fbAutoRequestBrightness_TON	: TOF;
	bInitTimeOut				: BOOL;
	fbInitTimeOut				: ARRAY [1.. nNumberOfSensors] OF TON;
	nIdxScan					: BYTE;
	nPirIdxOn					: BYTE;
	nBrightnessIdx				: BYTE;
	fBrightness_1				: REAL;
	fBrightness_2				: REAL;
	fBrightness_3				: REAL;
	fBrightness_4				: REAL;
	bInitDone					: BOOL;
	bInitScalesDone				: BOOL;
	
	nCheckIdx: INT;
END_VAR
VAR_IN_OUT
	stPirSensorData				: ST_DALI_Sensor;
	arrSensorScales				: ARRAY [1.. 10] OF ST_DALI_SensorScaleMode;
END_VAR

VAR CONSTANT
	nNumberOfSensors: BYTE := 4;
END_VAR

arrEsylux_PD_C[1].ipDALICommunication := ipCommunication;
arrEsylux_PD_C[2].ipDALICommunication := ipCommunication;
arrEsylux_PD_C[3].ipDALICommunication := ipCommunication;
arrEsylux_PD_C[4].ipDALICommunication := ipCommunication;

IF NOT bInitScalesDone THEN
	FOR nCheckIdx:= 1 TO 10 DO
		IF arrSensorScales[nCheckIdx].fMeassureMaxSensor = 0 THEN
			arrSensorScales[nCheckIdx].fMeassureMaxSensor := 1;
		END_IF
		IF arrSensorScales[nCheckIdx].fReadMaxSensor = 0 THEN
			arrSensorScales[nCheckIdx].fReadMaxSensor := 1;
		END_IF
	END_FOR
	bInitScalesDone := TRUE;
END_IF

IF ipCommunication <> 0 THEN
	A_ESYLux_4Pcs();
END_IF

ACTION A_ESYLux_4Pcs:


FOR nIdxScan := 1 TO nNumberOfSensors DO
	//Setup parameters
	//Setup Motion part of sensor (Instance 0)
	arrEsylux_PD_C[nIdxScan].bEnableOccupancy := TRUE;
	arrEsylux_PD_C[nIdxScan].eEventPriorityOccupancy:= eEventPriorityOccupancy;
	arrEsylux_PD_C[nIdxScan].nHoldTimerOccupancy := nHoldTimerOccupancy ;
	arrEsylux_PD_C[nIdxScan].nDeadtimeTimerOccupancy:= 	nDeadtimeTimerOccupancy;
	arrEsylux_PD_C[nIdxScan].nReportTimerOccupancy:= nReportTimerOccupancy;
	arrEsylux_PD_C[nIdxScan].nSensitivityOccupancy:= 100;
	
	//Setup Brightness part of sensor (Instance 1)
	arrEsylux_PD_C[nIdxScan].bEnableBrightness:= bEnableBrightness;
	arrEsylux_PD_C[nIdxScan].eEventPriorityBrightness:= eEventPriorityBrightness;
	arrEsylux_PD_C[nIdxScan].nDeadtimeTimerBrightness:= nDeadtimeTimerBrightness;
	arrEsylux_PD_C[nIdxScan].nHysteresisBrightness:= nHysteresisBrightness;
	arrEsylux_PD_C[nIdxScan].nHysteresisMinBrightness:= nHysteresisMinBrightness;
	arrEsylux_PD_C[nIdxScan].nReportTimerBrightness:= nReportTimerBrightness;

	arrEsylux_PD_C[nIdxScan].bModeLED:= bModeLED;
	arrEsylux_PD_C[nIdxScan].nBrightnessLED:= nBrightnessLED;
	
		
		
	//Calculate delay time for init sensor
	arrtDelayTime[nIdxScan] := INT_TO_TIME((BYTE_TO_INT((byShrtAdr + nIdxScan)-1) * 400));	
	arrDelaySetupDALIDevice[nIdxScan](IN:= bInitialize , PT:=arrtDelayTime[nIdxScan] , Q=> , ET=> );	
		
	IF arrDelaySetupDALIDevice[nIdxScan].q AND NOT GVL_DALI.arrbBlockDTR[DALI_LINE_NUM] AND NOT (arrInitDone[nIdxScan] OR arrInitErr[nIdxScan]) THEN
		arrInitSensor[nIdxScan]:= TRUE;
		GVL_DALI.arrbBlockDTR[DALI_LINE_NUM]:= TRUE;
	END_IF
	
	bQueryBrightness:= stPirSensorData.bQueryBrightness OR NOT bAutoRead;
	
	fbAutoRequestBrightness_TON(IN:= NOT fbAutoRequestBrightness_TON.Q  AND NOT stPirSensorData.bQueryBrightness , PT:= (arrtDelayTime[nIdxScan] + T#12M) , Q=>bAutoRead , ET=> );
	
	bQueryOccupancy:= NOT bAutoRead OR stPirSensorData.bQueryBrightness;
	
	arrEsylux_PD_C[nIdxScan](
		bError=> , 
		ipResultMessage=> , 
		bInitialize:=  arrInitSensor[nIdxScan], 
		nShortAddress:= (byShrtAdr + nIdxScan)-1 , 
		nOptions:= , 
		bQueryOccupancy:= bQueryOccupancy, 
		bQueryBrightness:= bQueryBrightness, 
		bCancelHoldTimerOccupancy:= bCancelHoldTimerOccupancy, 
		bInitializing=> arrInitializing[nIdxScan] , 
		bReadingOccupancy=> , 
		bReadingBrightness=> , 
		bOccupied=> , 
		nBrightnessLevel=> );
	
	arrInitDone_FTrig[nIdxScan](CLK:=arrInitializing[nIdxScan] );	
		IF arrInitDone_FTrig[nIdxScan].Q THEN
			IF NOT bInitTimeOut THEN
				arrInitDone[nIdxScan] := TRUE;
				GVL_DALI.arrbBlockDTR[DALI_LINE_NUM]:= FALSE;
			ELSE
				arrInitErr[nIdxScan] := TRUE;
				GVL_DALI.arrbBlockDTR[DALI_LINE_NUM]:= FALSE;
			END_IF
		END_IF
		
	fbInitTimeOut[nIdxScan](IN:=arrInitSensor[nIdxScan] AND NOT arrInitDone[nIdxScan], PT:= T#10S); 
	
	IF fbInitTimeOut[nIdxScan].Q THEN
		arrInitErr[nIdxScan] := TRUE;
		GVL_DALI.arrbBlockDTR[DALI_LINE_NUM]:= FALSE;
	END_IF
END_FOR

stPirSensorData.bPrc:= FALSE;
FOR nPirIdxOn:= 1 TO nNumberOfSensors DO
	IF arrEsylux_PD_C[nPirIdxOn].bOccupied THEN
		stPirSensorData.bPrc:= TRUE;
		EXIT;
	END_IF
END_FOR

stPirSensorData.bBrightnessRead:= arrEsylux_PD_C[1].bReadingBrightness OR arrEsylux_PD_C[2].bReadingBrightness OR arrEsylux_PD_C[3].bReadingBrightness OR arrEsylux_PD_C[4].bReadingBrightness;

fBrightness_1:= F_fScale(0, arrSensorScales[1].fReadMaxSensor, 0, arrSensorScales[1].fMeassureMaxSensor, 0, arrEsylux_PD_C[1].nBrightnessLevel);
fBrightness_2:= F_fScale(0, arrSensorScales[2].fReadMaxSensor, 0, arrSensorScales[2].fMeassureMaxSensor, 0, arrEsylux_PD_C[2].nBrightnessLevel);
fBrightness_3:= F_fScale(0, arrSensorScales[3].fReadMaxSensor, 0, arrSensorScales[3].fMeassureMaxSensor, 0, arrEsylux_PD_C[3].nBrightnessLevel);
fBrightness_4:= F_fScale(0, arrSensorScales[4].fReadMaxSensor, 0, arrSensorScales[4].fMeassureMaxSensor, 0, arrEsylux_PD_C[4].nBrightnessLevel);


IF fBrightness_1 <> 0 THEN
	stPirSensorData.fBrightness:= fBrightness_1;
END_IF
IF fBrightness_2 <> 0 THEN
	stPirSensorData.fBrightness:= MIN(fBrightness_2, stPirSensorData.fBrightness);
END_IF
IF fBrightness_3 <> 0 THEN
	stPirSensorData.fBrightness:=  MIN(fBrightness_3, stPirSensorData.fBrightness);
END_IF
IF fBrightness_4 <> 0 THEN
	stPirSensorData.fBrightness:=  MIN(fBrightness_4, stPirSensorData.fBrightness);
END_IF

IF NOT bInitialize THEN
	FOR nIdxScan := 1 TO nNumberOfSensors DO
		arrInitSensor[nIdxScan]:= FALSE;
		fbInitTimeOut[nIdxScan](IN:= FALSE);
		arrInitDone[nIdxScan] := FALSE;
		arrInitErr[nIdxScan] := FALSE;
	END_FOR
END_IF
END_ACTION

END_FUNCTION_BLOCK

// POUs/DALI/DALI_Devices/ESYLux/FB_DALI_ESYLux_5Pcs
FUNCTION_BLOCK FB_DALI_ESYLux_5Pcs
VAR_INPUT
	byShrtAdr					: BYTE;
	bInitialize					: BOOL := TRUE;
	ipCommunication				: I_DALICommunication;
	DALI_LINE_NUM				: INT := 1;	
END_VAR
VAR_OUTPUT
	arrInitErr: ARRAY [1.. nNumberOfSensors] OF BOOL;
	arrInitDone: ARRAY [1.. nNumberOfSensors] OF BOOL;
END_VAR
VAR
	arrEsylux_PD_C				: ARRAY [1.. nNumberOfSensors] OF FB_DALI_Esylux_PD_C_360_BMS(0);
	
	arrDelaySetupDALIDevice		: ARRAY [1.. nNumberOfSensors] Of TON;
	arrtDelayTime				: ARRAY [1.. nNumberOfSensors] OF TIME;
	arrInitSensor				: ARRAY [1.. nNumberOfSensors] OF BOOL;
	arrInitDone_FTrig			: ARRAY [1.. nNumberOfSensors] OF F_TRIG;
	arrInitializing				: ARRAY [1.. nNumberOfSensors] OF BOOL;

	bQueryBrightness 			: BOOL;
	bQueryOccupancy				: BOOL;

	eEventPriorityOccupancy		: E_DALIEventPriority := E_DALIEVENTPRIORITY.Middle;
	nHoldTimerOccupancy			: UINT := 5;
	nReportTimerOccupancy		: BYTE := 120; // Value in s, Preset manufacturer value
	nDeadtimeTimerOccupancy		: WORD := 100; // Value in ms, Predefined Value of DALI Standard
	bCancelHoldTimerOccupancy	: BOOL;
	nSensitivityOccupancy		: BYTE := 95; //setting Sensivity 0 = Low 100 = Max
	
	bEnableBrightness			: BOOL := FALSE;
	eEventPriorityBrightness	: E_DALIEventPriority := E_DALIEVENTPRIORITY.MiddleLow;
	nDeadtimeTimerBrightness	: WORD := 1500; // Value in ms, Predefined Value of DALI Standard
	nHysteresisBrightness		: BYTE := 5; // Value in %
	nHysteresisMinBrightness	: BYTE := 40; // Absolute Value, depending on the manufacturer specific resolution
	nReportTimerBrightness		: BYTE := 30; // Value in s, Preset manufacturer value

	bModeLED					: BOOL := FALSE; //LED mode: FALSE: LED disabled, TRUE: LED enabled
	nBrightnessLED				: USINT := 50; //LED brightness (5...100 %).

	bAutoRead					: BOOL;
	fbAutoRequestBrightness_TON	: TOF;
	bInitTimeOut				: BOOL;
	fbInitTimeOut				: ARRAY [1.. nNumberOfSensors] OF TON;
	nIdxScan					: BYTE;
	nPirIdxOn					: BYTE;
	nBrightnessIdx				: BYTE;
	fBrightness_1				: REAL;
	fBrightness_2				: REAL;
	fBrightness_3				: REAL;
	fBrightness_4				: REAL;
	fBrightness_5				: REAL;
	bInitDone					: BOOL;
	bInitScalesDone				: BOOL;
	
	nCheckIdx: INT;
END_VAR
VAR_IN_OUT
	stPirSensorData				: ST_DALI_Sensor;
	arrSensorScales				: ARRAY [1.. 10] OF ST_DALI_SensorScaleMode;
END_VAR

VAR CONSTANT
	nNumberOfSensors: BYTE := 5;
END_VAR

arrEsylux_PD_C[1].ipDALICommunication := ipCommunication;
arrEsylux_PD_C[2].ipDALICommunication := ipCommunication;
arrEsylux_PD_C[3].ipDALICommunication := ipCommunication;
arrEsylux_PD_C[4].ipDALICommunication := ipCommunication;
arrEsylux_PD_C[5].ipDALICommunication := ipCommunication;

IF NOT bInitScalesDone THEN
	FOR nCheckIdx:= 1 TO 10 DO
		IF arrSensorScales[nCheckIdx].fMeassureMaxSensor = 0 THEN
			arrSensorScales[nCheckIdx].fMeassureMaxSensor := 1;
		END_IF
		IF arrSensorScales[nCheckIdx].fReadMaxSensor = 0 THEN
			arrSensorScales[nCheckIdx].fReadMaxSensor := 1;
		END_IF
	END_FOR
	bInitScalesDone := TRUE;
END_IF

IF ipCommunication <> 0 THEN
	A_ESYLux_5Pcs();
END_IF

ACTION A_ESYLux_5Pcs:


FOR nIdxScan := 1 TO nNumberOfSensors DO
	//Setup parameters
	//Setup Motion part of sensor (Instance 0)
	arrEsylux_PD_C[nIdxScan].bEnableOccupancy := TRUE;
	arrEsylux_PD_C[nIdxScan].eEventPriorityOccupancy:= eEventPriorityOccupancy;
	arrEsylux_PD_C[nIdxScan].nHoldTimerOccupancy := nHoldTimerOccupancy ;
	arrEsylux_PD_C[nIdxScan].nDeadtimeTimerOccupancy:= 	nDeadtimeTimerOccupancy;
	arrEsylux_PD_C[nIdxScan].nReportTimerOccupancy:= nReportTimerOccupancy;
	arrEsylux_PD_C[nIdxScan].nSensitivityOccupancy:= 100;
	
	//Setup Brightness part of sensor (Instance 1)
	arrEsylux_PD_C[nIdxScan].bEnableBrightness:= bEnableBrightness;
	arrEsylux_PD_C[nIdxScan].eEventPriorityBrightness:= eEventPriorityBrightness;
	arrEsylux_PD_C[nIdxScan].nDeadtimeTimerBrightness:= nDeadtimeTimerBrightness;
	arrEsylux_PD_C[nIdxScan].nHysteresisBrightness:= nHysteresisBrightness;
	arrEsylux_PD_C[nIdxScan].nHysteresisMinBrightness:= nHysteresisMinBrightness;
	arrEsylux_PD_C[nIdxScan].nReportTimerBrightness:= nReportTimerBrightness;

	arrEsylux_PD_C[nIdxScan].bModeLED:= bModeLED;
	arrEsylux_PD_C[nIdxScan].nBrightnessLED:= nBrightnessLED;
	
		
		
	//Calculate delay time for init sensor
	arrtDelayTime[nIdxScan] := INT_TO_TIME((BYTE_TO_INT((byShrtAdr + nIdxScan)-1) * 400));	
	arrDelaySetupDALIDevice[nIdxScan](IN:= bInitialize , PT:=arrtDelayTime[nIdxScan] , Q=> , ET=> );	
		
	IF arrDelaySetupDALIDevice[nIdxScan].q AND NOT GVL_DALI.arrbBlockDTR[DALI_LINE_NUM] AND NOT (arrInitDone[nIdxScan] OR arrInitErr[nIdxScan]) THEN
		arrInitSensor[nIdxScan]:= TRUE;
		GVL_DALI.arrbBlockDTR[DALI_LINE_NUM]:= TRUE;
	END_IF
	
	bQueryBrightness:= stPirSensorData.bQueryBrightness OR NOT bAutoRead;
	
	fbAutoRequestBrightness_TON(IN:= NOT fbAutoRequestBrightness_TON.Q  AND NOT stPirSensorData.bQueryBrightness , PT:= (arrtDelayTime[nIdxScan] + T#12M) , Q=>bAutoRead , ET=> );
	
	bQueryOccupancy:= NOT bAutoRead OR stPirSensorData.bQueryBrightness;
	
	arrEsylux_PD_C[nIdxScan](
		bError=> , 
		ipResultMessage=> , 
		bInitialize:=  arrInitSensor[nIdxScan], 
		nShortAddress:= (byShrtAdr + nIdxScan)-1 , 
		nOptions:= , 
		bQueryOccupancy:= bQueryOccupancy, 
		bQueryBrightness:= bQueryBrightness, 
		bCancelHoldTimerOccupancy:= bCancelHoldTimerOccupancy, 
		bInitializing=> arrInitializing[nIdxScan] , 
		bReadingOccupancy=> , 
		bReadingBrightness=> , 
		bOccupied=> , 
		nBrightnessLevel=> );
	
	arrInitDone_FTrig[nIdxScan](CLK:=arrInitializing[nIdxScan] );	
		IF arrInitDone_FTrig[nIdxScan].Q THEN
			IF NOT bInitTimeOut THEN
				arrInitDone[nIdxScan] := TRUE;
				GVL_DALI.arrbBlockDTR[DALI_LINE_NUM]:= FALSE;
			ELSE
				arrInitErr[nIdxScan] := TRUE;
				GVL_DALI.arrbBlockDTR[DALI_LINE_NUM]:= FALSE;
			END_IF
		END_IF
		
	fbInitTimeOut[nIdxScan](IN:=arrInitSensor[nIdxScan] AND NOT arrInitDone[nIdxScan], PT:= T#10S); 
	
	IF fbInitTimeOut[nIdxScan].Q THEN
		arrInitErr[nIdxScan] := TRUE;
		GVL_DALI.arrbBlockDTR[DALI_LINE_NUM]:= FALSE;
	END_IF
END_FOR

stPirSensorData.bPrc:= FALSE;
FOR nPirIdxOn:= 1 TO nNumberOfSensors DO
	IF arrEsylux_PD_C[nPirIdxOn].bOccupied THEN
		stPirSensorData.bPrc:= TRUE;
		EXIT;
	END_IF
END_FOR

stPirSensorData.bBrightnessRead:= arrEsylux_PD_C[1].bReadingBrightness OR arrEsylux_PD_C[2].bReadingBrightness OR arrEsylux_PD_C[3].bReadingBrightness OR arrEsylux_PD_C[4].bReadingBrightness OR arrEsylux_PD_C[5].bReadingBrightness;

fBrightness_1:= F_fScale(0, arrSensorScales[1].fReadMaxSensor, 0, arrSensorScales[1].fMeassureMaxSensor, 0, arrEsylux_PD_C[1].nBrightnessLevel);
fBrightness_2:= F_fScale(0, arrSensorScales[2].fReadMaxSensor, 0, arrSensorScales[2].fMeassureMaxSensor, 0, arrEsylux_PD_C[2].nBrightnessLevel);
fBrightness_3:= F_fScale(0, arrSensorScales[3].fReadMaxSensor, 0, arrSensorScales[3].fMeassureMaxSensor, 0, arrEsylux_PD_C[3].nBrightnessLevel);
fBrightness_4:= F_fScale(0, arrSensorScales[4].fReadMaxSensor, 0, arrSensorScales[4].fMeassureMaxSensor, 0, arrEsylux_PD_C[4].nBrightnessLevel);
fBrightness_5:= F_fScale(0, arrSensorScales[5].fReadMaxSensor, 0, arrSensorScales[5].fMeassureMaxSensor, 0, arrEsylux_PD_C[5].nBrightnessLevel);


IF fBrightness_1 <> 0 THEN
	stPirSensorData.fBrightness:= fBrightness_1;
END_IF
IF fBrightness_2 <> 0 THEN
	stPirSensorData.fBrightness:= MIN(fBrightness_2, stPirSensorData.fBrightness);
END_IF
IF fBrightness_3 <> 0 THEN
	stPirSensorData.fBrightness:=  MIN(fBrightness_3, stPirSensorData.fBrightness);
END_IF
IF fBrightness_4 <> 0 THEN
	stPirSensorData.fBrightness:=  MIN(fBrightness_4, stPirSensorData.fBrightness);
END_IF
IF fBrightness_5 <> 0 THEN
	stPirSensorData.fBrightness:=  MIN(fBrightness_5, stPirSensorData.fBrightness);
END_IF


IF NOT bInitialize THEN
	FOR nIdxScan := 1 TO nNumberOfSensors DO
		arrInitSensor[nIdxScan]:= FALSE;
		fbInitTimeOut[nIdxScan](IN:= FALSE);
		arrInitDone[nIdxScan] := FALSE;
		arrInitErr[nIdxScan] := FALSE;
	END_FOR
END_IF
END_ACTION

END_FUNCTION_BLOCK

// POUs/DALI/DALI_Devices/ESYLux/FB_DALI_ESYLux_6Pcs
FUNCTION_BLOCK FB_DALI_ESYLux_6Pcs
VAR_INPUT
	byShrtAdr					: BYTE;
	bInitialize					: BOOL := TRUE;
	ipCommunication				: I_DALICommunication;
	DALI_LINE_NUM				: INT := 1;	
END_VAR
VAR_OUTPUT
	arrInitErr: ARRAY [1.. nNumberOfSensors] OF BOOL;
	arrInitDone: ARRAY [1.. nNumberOfSensors] OF BOOL;
END_VAR
VAR
	arrEsylux_PD_C				: ARRAY [1.. nNumberOfSensors] OF FB_DALI_Esylux_PD_C_360_BMS(0);
	
	arrDelaySetupDALIDevice		: ARRAY [1.. nNumberOfSensors] Of TON;
	arrtDelayTime				: ARRAY [1.. nNumberOfSensors] OF TIME;
	arrInitSensor				: ARRAY [1.. nNumberOfSensors] OF BOOL;
	arrInitDone_FTrig			: ARRAY [1.. nNumberOfSensors] OF F_TRIG;
	arrInitializing				: ARRAY [1.. nNumberOfSensors] OF BOOL;

	bQueryBrightness 			: BOOL;
	bQueryOccupancy				: BOOL;

	eEventPriorityOccupancy		: E_DALIEventPriority := E_DALIEVENTPRIORITY.Middle;
	nHoldTimerOccupancy			: UINT := 5;
	nReportTimerOccupancy		: BYTE := 120; // Value in s, Preset manufacturer value
	nDeadtimeTimerOccupancy		: WORD := 100; // Value in ms, Predefined Value of DALI Standard
	bCancelHoldTimerOccupancy	: BOOL;
	nSensitivityOccupancy		: BYTE := 95; //setting Sensivity 0 = Low 100 = Max
	
	bEnableBrightness			: BOOL := FALSE;
	eEventPriorityBrightness	: E_DALIEventPriority := E_DALIEVENTPRIORITY.MiddleLow;
	nDeadtimeTimerBrightness	: WORD := 1500; // Value in ms, Predefined Value of DALI Standard
	nHysteresisBrightness		: BYTE := 5; // Value in %
	nHysteresisMinBrightness	: BYTE := 40; // Absolute Value, depending on the manufacturer specific resolution
	nReportTimerBrightness		: BYTE := 30; // Value in s, Preset manufacturer value

	bModeLED					: BOOL := FALSE; //LED mode: FALSE: LED disabled, TRUE: LED enabled
	nBrightnessLED				: USINT := 50; //LED brightness (5...100 %).

	bAutoRead					: BOOL;
	fbAutoRequestBrightness_TON	: TOF;
	bInitTimeOut				: BOOL;
	fbInitTimeOut				: ARRAY [1.. nNumberOfSensors] OF TON;
	nIdxScan					: BYTE;
	nPirIdxOn					: BYTE;
	nBrightnessIdx				: BYTE;
	fBrightness_1				: REAL;
	fBrightness_2				: REAL;
	fBrightness_3				: REAL;
	fBrightness_4				: REAL;
	fBrightness_5				: REAL;
	fBrightness_6				: REAL;
	bInitDone					: BOOL;
	bInitScalesDone				: BOOL;
	
	nCheckIdx: INT;
END_VAR
VAR_IN_OUT
	stPirSensorData				: ST_DALI_Sensor;
	arrSensorScales				: ARRAY [1.. 10] OF ST_DALI_SensorScaleMode;
END_VAR

VAR CONSTANT
	nNumberOfSensors: BYTE := 6;
END_VAR

arrEsylux_PD_C[1].ipDALICommunication := ipCommunication;
arrEsylux_PD_C[2].ipDALICommunication := ipCommunication;
arrEsylux_PD_C[3].ipDALICommunication := ipCommunication;
arrEsylux_PD_C[4].ipDALICommunication := ipCommunication;
arrEsylux_PD_C[5].ipDALICommunication := ipCommunication;
arrEsylux_PD_C[6].ipDALICommunication := ipCommunication;

IF NOT bInitScalesDone THEN
	FOR nCheckIdx:= 1 TO 10 DO
		IF arrSensorScales[nCheckIdx].fMeassureMaxSensor = 0 THEN
			arrSensorScales[nCheckIdx].fMeassureMaxSensor := 1;
		END_IF
		IF arrSensorScales[nCheckIdx].fReadMaxSensor = 0 THEN
			arrSensorScales[nCheckIdx].fReadMaxSensor := 1;
		END_IF
	END_FOR
	bInitScalesDone := TRUE;
END_IF

IF ipCommunication <> 0 THEN
	A_ESYLux_6Pcs();
END_IF

ACTION A_ESYLux_6Pcs:


FOR nIdxScan := 1 TO nNumberOfSensors DO
	//Setup parameters
	//Setup Motion part of sensor (Instance 0)
	arrEsylux_PD_C[nIdxScan].bEnableOccupancy := TRUE;
	arrEsylux_PD_C[nIdxScan].eEventPriorityOccupancy:= eEventPriorityOccupancy;
	arrEsylux_PD_C[nIdxScan].nHoldTimerOccupancy := nHoldTimerOccupancy ;
	arrEsylux_PD_C[nIdxScan].nDeadtimeTimerOccupancy:= 	nDeadtimeTimerOccupancy;
	arrEsylux_PD_C[nIdxScan].nReportTimerOccupancy:= nReportTimerOccupancy;
	arrEsylux_PD_C[nIdxScan].nSensitivityOccupancy:= 100;
	
	//Setup Brightness part of sensor (Instance 1)
	arrEsylux_PD_C[nIdxScan].bEnableBrightness:= bEnableBrightness;
	arrEsylux_PD_C[nIdxScan].eEventPriorityBrightness:= eEventPriorityBrightness;
	arrEsylux_PD_C[nIdxScan].nDeadtimeTimerBrightness:= nDeadtimeTimerBrightness;
	arrEsylux_PD_C[nIdxScan].nHysteresisBrightness:= nHysteresisBrightness;
	arrEsylux_PD_C[nIdxScan].nHysteresisMinBrightness:= nHysteresisMinBrightness;
	arrEsylux_PD_C[nIdxScan].nReportTimerBrightness:= nReportTimerBrightness;

	arrEsylux_PD_C[nIdxScan].bModeLED:= bModeLED;
	arrEsylux_PD_C[nIdxScan].nBrightnessLED:= nBrightnessLED;
	
		
		
	//Calculate delay time for init sensor
	arrtDelayTime[nIdxScan] := INT_TO_TIME((BYTE_TO_INT((byShrtAdr + nIdxScan)-1) * 400));	
	arrDelaySetupDALIDevice[nIdxScan](IN:= bInitialize , PT:=arrtDelayTime[nIdxScan] , Q=> , ET=> );	
		
	IF arrDelaySetupDALIDevice[nIdxScan].q AND NOT GVL_DALI.arrbBlockDTR[DALI_LINE_NUM] AND NOT (arrInitDone[nIdxScan] OR arrInitErr[nIdxScan]) THEN
		arrInitSensor[nIdxScan]:= TRUE;
		GVL_DALI.arrbBlockDTR[DALI_LINE_NUM]:= TRUE;
	END_IF
	
	bQueryBrightness:= stPirSensorData.bQueryBrightness OR NOT bAutoRead;
	
	fbAutoRequestBrightness_TON(IN:= NOT fbAutoRequestBrightness_TON.Q  AND NOT stPirSensorData.bQueryBrightness , PT:= (arrtDelayTime[nIdxScan] + T#12M) , Q=>bAutoRead , ET=> );
	
	bQueryOccupancy:= NOT bAutoRead OR stPirSensorData.bQueryBrightness;
	
	arrEsylux_PD_C[nIdxScan](
		bError=> , 
		ipResultMessage=> , 
		bInitialize:=  arrInitSensor[nIdxScan], 
		nShortAddress:= (byShrtAdr + nIdxScan)-1 , 
		nOptions:= , 
		bQueryOccupancy:= bQueryOccupancy, 
		bQueryBrightness:= bQueryBrightness, 
		bCancelHoldTimerOccupancy:= bCancelHoldTimerOccupancy, 
		bInitializing=> arrInitializing[nIdxScan] , 
		bReadingOccupancy=> , 
		bReadingBrightness=> , 
		bOccupied=> , 
		nBrightnessLevel=> );
	
	arrInitDone_FTrig[nIdxScan](CLK:=arrInitializing[nIdxScan] );	
		IF arrInitDone_FTrig[nIdxScan].Q THEN
			IF NOT bInitTimeOut THEN
				arrInitDone[nIdxScan] := TRUE;
				GVL_DALI.arrbBlockDTR[DALI_LINE_NUM]:= FALSE;
			ELSE
				arrInitErr[nIdxScan] := TRUE;
				GVL_DALI.arrbBlockDTR[DALI_LINE_NUM]:= FALSE;
			END_IF
		END_IF
		
	fbInitTimeOut[nIdxScan](IN:=arrInitSensor[nIdxScan] AND NOT arrInitDone[nIdxScan], PT:= T#10S); 
	
	IF fbInitTimeOut[nIdxScan].Q THEN
		arrInitErr[nIdxScan] := TRUE;
		GVL_DALI.arrbBlockDTR[DALI_LINE_NUM]:= FALSE;
	END_IF
END_FOR

stPirSensorData.bPrc:= FALSE;
FOR nPirIdxOn:= 1 TO nNumberOfSensors DO
	IF arrEsylux_PD_C[nPirIdxOn].bOccupied THEN
		stPirSensorData.bPrc:= TRUE;
		EXIT;
	END_IF
END_FOR

stPirSensorData.bBrightnessRead:= arrEsylux_PD_C[1].bReadingBrightness 
									OR arrEsylux_PD_C[2].bReadingBrightness 
										OR arrEsylux_PD_C[3].bReadingBrightness 
											OR arrEsylux_PD_C[4].bReadingBrightness 
												OR arrEsylux_PD_C[5].bReadingBrightness 
													OR arrEsylux_PD_C[6].bReadingBrightness;

fBrightness_1:= F_fScale(0, arrSensorScales[1].fReadMaxSensor, 0, arrSensorScales[1].fMeassureMaxSensor, 0, arrEsylux_PD_C[1].nBrightnessLevel);
fBrightness_2:= F_fScale(0, arrSensorScales[2].fReadMaxSensor, 0, arrSensorScales[2].fMeassureMaxSensor, 0, arrEsylux_PD_C[2].nBrightnessLevel);
fBrightness_3:= F_fScale(0, arrSensorScales[3].fReadMaxSensor, 0, arrSensorScales[3].fMeassureMaxSensor, 0, arrEsylux_PD_C[3].nBrightnessLevel);
fBrightness_4:= F_fScale(0, arrSensorScales[4].fReadMaxSensor, 0, arrSensorScales[4].fMeassureMaxSensor, 0, arrEsylux_PD_C[4].nBrightnessLevel);
fBrightness_5:= F_fScale(0, arrSensorScales[5].fReadMaxSensor, 0, arrSensorScales[5].fMeassureMaxSensor, 0, arrEsylux_PD_C[5].nBrightnessLevel);
fBrightness_6:= F_fScale(0, arrSensorScales[6].fReadMaxSensor, 0, arrSensorScales[6].fMeassureMaxSensor, 0, arrEsylux_PD_C[6].nBrightnessLevel);


IF fBrightness_1 <> 0 THEN
	stPirSensorData.fBrightness:= fBrightness_1;
END_IF
IF fBrightness_2 <> 0 THEN
	stPirSensorData.fBrightness:= MIN(fBrightness_2, stPirSensorData.fBrightness);
END_IF
IF fBrightness_3 <> 0 THEN
	stPirSensorData.fBrightness:=  MIN(fBrightness_3, stPirSensorData.fBrightness);
END_IF
IF fBrightness_4 <> 0 THEN
	stPirSensorData.fBrightness:=  MIN(fBrightness_4, stPirSensorData.fBrightness);
END_IF
IF fBrightness_5 <> 0 THEN
	stPirSensorData.fBrightness:=  MIN(fBrightness_5, stPirSensorData.fBrightness);
END_IF
IF fBrightness_6 <> 0 THEN
	stPirSensorData.fBrightness:=  MIN(fBrightness_6, stPirSensorData.fBrightness);
END_IF

IF NOT bInitialize THEN
	FOR nIdxScan := 1 TO nNumberOfSensors DO
		arrInitSensor[nIdxScan]:= FALSE;
		fbInitTimeOut[nIdxScan](IN:= FALSE);
		arrInitDone[nIdxScan] := FALSE;
		arrInitErr[nIdxScan] := FALSE;
	END_FOR
END_IF
END_ACTION

END_FUNCTION_BLOCK

// POUs/DALI/DALI_Devices/Glamox/FB_DALI_GlamoxButtons
FUNCTION_BLOCK FB_DALI_GlamoxButtons
VAR_INPUT
	byShrtAdr				: BYTE;
	bInitialize				: BOOL := TRUE;
	ipCommunication			: I_DALICommunication;
	DALI_LINE_NUM			: INT := 1;	
	stGlamoxSetup			: ST_GlamoxSetup;		
END_VAR
VAR_OUTPUT
	arrButtons				: ARRAY [1..8] OF ST_DALIButton;
END_VAR
		
VAR
	fbButtons 				: FB_DALI_Glamox_LMS_PB8_SwitchPanel(0) ;

	arrQueryInput 			: ARRAY [1..8] OF BOOL;
	arrReadingInput 		: ARRAY [1..8] OF BOOL;
	arrPushButtonEvent 		: ARRAY [1..8] OF WORD; (* Bit 0 - Push button released.
									 Bit 1 - Push button pressed..
									 Bit 2 - Short keystroke.
									 Bit 3 - Double keystroke.
									 Bit 4 - Start long keystroke.
									 Bit 5 - Repeat long keystroke.
									 Bit 6 - Stop long keystroke.
									 Bit 7 - Push button free again; was previously blocked.
									 Bit 8 - Push button blocked. *)

	fbDelaySetupDALIDevice	: TON;
	tDelayTime				: TIME;
	bInitSensor				: BOOL;
	fbInitDone				: F_TRIG;
	bInitDone				: BOOL;
	bInitErr				: BOOL;
	bInitializing			: BOOL;
	bInitTimeOut			: BOOL;
	fbInitTimeOut			: TON;
END_VAR

fbButtons.ipDALICommunication:= ipCommunication ;

	fbButtons.bEnablePushButton1:= stGlamoxSetup.arrEnablePushButton[1];
	fbButtons.bEnablePushButton2:= stGlamoxSetup.arrEnablePushButton[2];
	fbButtons.bEnablePushButton3:= stGlamoxSetup.arrEnablePushButton[3];
	fbButtons.bEnablePushButton4:= stGlamoxSetup.arrEnablePushButton[4];
	fbButtons.bEnablePushButton5:= stGlamoxSetup.arrEnablePushButton[5];
	fbButtons.bEnablePushButton6:= stGlamoxSetup.arrEnablePushButton[6];
	fbButtons.bEnablePushButton7:= stGlamoxSetup.arrEnablePushButton[7];
	fbButtons.bEnablePushButton8:= stGlamoxSetup.arrEnablePushButton[8];
	
	fbButtons.eEventPriorityPushButton1:= stGlamoxSetup.arrEventPriorityPushButton[1];
	fbButtons.eEventPriorityPushButton2:= stGlamoxSetup.arrEventPriorityPushButton[2];
	fbButtons.eEventPriorityPushButton3:= stGlamoxSetup.arrEventPriorityPushButton[3];
	fbButtons.eEventPriorityPushButton4:= stGlamoxSetup.arrEventPriorityPushButton[4];
	fbButtons.eEventPriorityPushButton5:= stGlamoxSetup.arrEventPriorityPushButton[5];
	fbButtons.eEventPriorityPushButton6:= stGlamoxSetup.arrEventPriorityPushButton[6];
	fbButtons.eEventPriorityPushButton7:= stGlamoxSetup.arrEventPriorityPushButton[7];
	fbButtons.eEventPriorityPushButton8:= stGlamoxSetup.arrEventPriorityPushButton[8];

	fbButtons.nDoubleTimerPushButton1 := stGlamoxSetup.nDoubleTimerPushButton;
	fbButtons.nDoubleTimerPushButton2:= stGlamoxSetup.nDoubleTimerPushButton;
	fbButtons.nDoubleTimerPushButton3:= stGlamoxSetup.nDoubleTimerPushButton;
	fbButtons.nDoubleTimerPushButton4:= stGlamoxSetup.nDoubleTimerPushButton;
	fbButtons.nDoubleTimerPushButton5:= stGlamoxSetup.nDoubleTimerPushButton;
	fbButtons.nDoubleTimerPushButton6:= stGlamoxSetup.nDoubleTimerPushButton;
	fbButtons.nDoubleTimerPushButton7:= stGlamoxSetup.nDoubleTimerPushButton;
	fbButtons.nDoubleTimerPushButton8:= stGlamoxSetup.nDoubleTimerPushButton;
	
	fbButtons.nEventFilterPushButton1 :=stGlamoxSetup.nEventFilterPushButton[1] ;
	fbButtons.nEventFilterPushButton2 :=stGlamoxSetup.nEventFilterPushButton[2] ;
	fbButtons.nEventFilterPushButton3 :=stGlamoxSetup.nEventFilterPushButton[3] ;
	fbButtons.nEventFilterPushButton4 :=stGlamoxSetup.nEventFilterPushButton[4] ;
	fbButtons.nEventFilterPushButton5 :=stGlamoxSetup.nEventFilterPushButton[5] ;
	fbButtons.nEventFilterPushButton6 :=stGlamoxSetup.nEventFilterPushButton[6] ;
	fbButtons.nEventFilterPushButton7 :=stGlamoxSetup.nEventFilterPushButton[7] ;
	fbButtons.nEventFilterPushButton8 :=stGlamoxSetup.nEventFilterPushButton[8] ;
	
	fbButtons.nRepeatTimerPushButton1 := stGlamoxSetup.nRepeatTimerPushButton;
	fbButtons.nRepeatTimerPushButton2 := stGlamoxSetup.nRepeatTimerPushButton;
	fbButtons.nRepeatTimerPushButton3 := stGlamoxSetup.nRepeatTimerPushButton;
	fbButtons.nRepeatTimerPushButton4 := stGlamoxSetup.nRepeatTimerPushButton;
	fbButtons.nRepeatTimerPushButton5 := stGlamoxSetup.nRepeatTimerPushButton;
	fbButtons.nRepeatTimerPushButton6 := stGlamoxSetup.nRepeatTimerPushButton;
	fbButtons.nRepeatTimerPushButton7 := stGlamoxSetup.nRepeatTimerPushButton;
	fbButtons.nRepeatTimerPushButton8 := stGlamoxSetup.nRepeatTimerPushButton;
	
	fbButtons.nShortTimerPushButton1 := stGlamoxSetup.nShortTimerPushButton ;
	fbButtons.nShortTimerPushButton2 := stGlamoxSetup.nShortTimerPushButton ;
	fbButtons.nShortTimerPushButton3 := stGlamoxSetup.nShortTimerPushButton ;
	fbButtons.nShortTimerPushButton4 := stGlamoxSetup.nShortTimerPushButton ;
	fbButtons.nShortTimerPushButton5 := stGlamoxSetup.nShortTimerPushButton ;
	fbButtons.nShortTimerPushButton6 := stGlamoxSetup.nShortTimerPushButton ;
	fbButtons.nShortTimerPushButton7 := stGlamoxSetup.nShortTimerPushButton ;
	fbButtons.nShortTimerPushButton8 := stGlamoxSetup.nShortTimerPushButton ;
	
	fbButtons.nStuckTimerPushButton1 := stGlamoxSetup.nStuckTimerPushButton ;
	fbButtons.nStuckTimerPushButton2 := stGlamoxSetup.nStuckTimerPushButton ;
	fbButtons.nStuckTimerPushButton3 := stGlamoxSetup.nStuckTimerPushButton ;
	fbButtons.nStuckTimerPushButton4 := stGlamoxSetup.nStuckTimerPushButton ;
	fbButtons.nStuckTimerPushButton5 := stGlamoxSetup.nStuckTimerPushButton ;
	fbButtons.nStuckTimerPushButton6 := stGlamoxSetup.nStuckTimerPushButton ;
	fbButtons.nStuckTimerPushButton7 := stGlamoxSetup.nStuckTimerPushButton ;
	fbButtons.nStuckTimerPushButton8 := stGlamoxSetup.nStuckTimerPushButton ;

//Calculate delay time for init sensor
tDelayTime := INT_TO_TIME((BYTE_TO_INT(byShrtAdr) * 400));	
fbDelaySetupDALIDevice(IN:= bInitialize , PT:=tDelayTime , Q=> , ET=> );	
	
IF fbDelaySetupDALIDevice.q AND NOT GVL_DALI.arrbBlockDTR[DALI_LINE_NUM] AND NOT (bInitDone OR bInitErr) THEN
	bInitDone := FALSE;
	bInitErr := FALSE;
	bInitSensor:= TRUE;
	GVL_DALI.arrbBlockDTR[DALI_LINE_NUM]:= TRUE;
END_IF

fbButtons(
	bError=> , 
	ipResultMessage=> , 
	bInitialize:= bInitSensor , 
	nShortAddress:= byShrtAdr, 
	nOptions:= , 
	bQueryInputValue1:= arrQueryInput[1], 
	bQueryInputValue2:= arrQueryInput[2], 
	bQueryInputValue3:= arrQueryInput[3], 
	bQueryInputValue4:= arrQueryInput[4], 
	bQueryInputValue5:= arrQueryInput[5], 
	bQueryInputValue6:= arrQueryInput[6], 
	bQueryInputValue7:= arrQueryInput[7], 
	bQueryInputValue8:= arrQueryInput[8], 
	bInitializing=> bInitializing, 
	bReadingInputValue1=> arrReadingInput[1] , 
	bReadingInputValue2=> arrReadingInput[2] , 
	bReadingInputValue3=> arrReadingInput[3] , 
	bReadingInputValue4=> arrReadingInput[4] , 
	bReadingInputValue5=> arrReadingInput[5] , 
	bReadingInputValue6=> arrReadingInput[6] , 
	bReadingInputValue7=> arrReadingInput[7] , 
	bReadingInputValue8=> arrReadingInput[8] , 
	nPushButton1Event=> arrPushButtonEvent[1], 
	nPushButton2Event=> arrPushButtonEvent[2], 
	nPushButton3Event=> arrPushButtonEvent[3], 
	nPushButton4Event=> arrPushButtonEvent[4], 
	nPushButton5Event=> arrPushButtonEvent[5], 
	nPushButton6Event=> arrPushButtonEvent[6], 
	nPushButton7Event=> arrPushButtonEvent[7], 
	nPushButton8Event=> arrPushButtonEvent[8]);
	
fbInitDone(CLK:=bInitSensor AND bInitializing );	
	IF fbInitDone.Q THEN
		IF NOT bInitTimeOut THEN
			bInitDone := TRUE;
			bInitErr := FALSE;
			GVL_DALI.arrbBlockDTR[DALI_LINE_NUM]:= FALSE;
		ELSE
			bInitErr := TRUE;
			GVL_DALI.arrbBlockDTR[DALI_LINE_NUM]:= FALSE;
		END_IF
	END_IF

fbInitTimeOut(IN:=bInitializing, PT:= T#15S); 

IF fbInitTimeOut.Q THEN
	bInitErr := TRUE;
	GVL_DALI.arrbBlockDTR[DALI_LINE_NUM]:= FALSE;
END_IF


IF NOT bInitialize THEN
		fbInitTimeOut(IN:= FALSE);
		bInitSensor:= FALSE;
		bInitDone := FALSE;
		bInitErr := FALSE;
END_IF	
	A_Sort_Event_Button1();
	A_Sort_Event_Button2();
	A_Sort_Event_Button3();
	A_Sort_Event_Button4();
	A_Sort_Event_Button5();
	A_Sort_Event_Button6();
	A_Sort_Event_Button7();
	A_Sort_Event_Button8();

ACTION A_Sort_Event_Button1:

IF arrPushButtonEvent[1].1 THEN
	arrButtons[1].bPressed:= TRUE;
	arrButtons[1].bReleased:= FALSE;
END_IF

IF arrPushButtonEvent[1].0 THEN
	arrButtons[1].bPressed:= FALSE;
	arrButtons[1].bReleased:= TRUE;
END_IF

IF arrPushButtonEvent[1].2 THEN
	arrButtons[1].bShortPress:= TRUE;
END_IF

IF arrPushButtonEvent[1].3 THEN
	arrButtons[1].bDoublePress:= TRUE;
END_IF

IF arrPushButtonEvent[1].4 THEN
	arrButtons[1].bLongPressStop:= FALSE;
	arrButtons[1].bLongPressStart:= TRUE;
	arrButtons[1].bLongPressRepeat:= FALSE;	
END_IF

arrButtons[1].bLongPressRepeat:= arrPushButtonEvent[1].5 ;

IF arrPushButtonEvent[1].6 THEN
	arrButtons[1].bLongPressStop:= TRUE;
	arrButtons[1].bLongPressStart:= FALSE;
	arrButtons[1].bLongPressRepeat:= FALSE;	
END_IF

IF arrPushButtonEvent[1].7 THEN
	arrButtons[1].bPressed:= FALSE;
	arrButtons[1].bReleased:= FALSE;
	arrButtons[1].bShortPress:= FALSE;
	arrButtons[1].bDoublePress:= FALSE;	
	arrButtons[1].bLongPressStart:= FALSE;
	arrButtons[1].bLongPressRepeat:= FALSE;	
	arrButtons[1].bLongPressStop:= FALSE;	
	arrButtons[1].bButtonFree := TRUE;
END_IF
END_ACTION

ACTION A_Sort_Event_Button2:

IF arrPushButtonEvent[2].1 THEN
	arrButtons[2].bPressed:= TRUE;
	arrButtons[2].bReleased:= FALSE;
END_IF

IF arrPushButtonEvent[2].0 THEN
	arrButtons[2].bPressed:= FALSE;
	arrButtons[2].bReleased:= TRUE;
END_IF

IF arrPushButtonEvent[2].2 THEN
	arrButtons[2].bShortPress:= TRUE;
END_IF

IF arrPushButtonEvent[2].3 THEN
	arrButtons[2].bDoublePress:= TRUE;
END_IF

IF arrPushButtonEvent[2].4 THEN
	arrButtons[2].bLongPressStop:= FALSE;
	arrButtons[2].bLongPressStart:= TRUE;
	arrButtons[2].bLongPressRepeat:= FALSE;	
END_IF

arrButtons[2].bLongPressRepeat:= arrPushButtonEvent[2].5 ;

IF arrPushButtonEvent[2].6 THEN
	arrButtons[2].bLongPressStop:= TRUE;
	arrButtons[2].bLongPressStart:= FALSE;
	arrButtons[2].bLongPressRepeat:= FALSE;	
END_IF

IF arrPushButtonEvent[2].7 THEN
	arrButtons[2].bPressed:= FALSE;
	arrButtons[2].bReleased:= FALSE;
	arrButtons[2].bShortPress:= FALSE;
	arrButtons[2].bDoublePress:= FALSE;	
	arrButtons[2].bLongPressStart:= FALSE;
	arrButtons[2].bLongPressRepeat:= FALSE;	
	arrButtons[2].bLongPressStop:= FALSE;	
	arrButtons[2].bButtonFree := TRUE;
END_IF
END_ACTION

ACTION A_Sort_Event_Button3:

IF arrPushButtonEvent[3].1 THEN
	arrButtons[3].bPressed:= TRUE;
	arrButtons[3].bReleased:= FALSE;
END_IF

IF arrPushButtonEvent[3].0 THEN
	arrButtons[3].bPressed:= FALSE;
	arrButtons[3].bReleased:= TRUE;
END_IF

IF arrPushButtonEvent[3].2 THEN
	arrButtons[3].bShortPress:= TRUE;
END_IF

IF arrPushButtonEvent[3].3 THEN
	arrButtons[3].bDoublePress:= TRUE;
END_IF

IF arrPushButtonEvent[3].4 THEN
	arrButtons[3].bLongPressStop:= FALSE;
	arrButtons[3].bLongPressStart:= TRUE;
	arrButtons[3].bLongPressRepeat:= FALSE;	
END_IF

arrButtons[3].bLongPressRepeat:= arrPushButtonEvent[3].5 ;

IF arrPushButtonEvent[3].6 THEN
	arrButtons[3].bLongPressStop:= TRUE;
	arrButtons[3].bLongPressStart:= FALSE;
	arrButtons[3].bLongPressRepeat:= FALSE;	
END_IF

IF arrPushButtonEvent[3].7 THEN
	arrButtons[3].bPressed:= FALSE;
	arrButtons[3].bReleased:= FALSE;
	arrButtons[3].bShortPress:= FALSE;
	arrButtons[3].bDoublePress:= FALSE;	
	arrButtons[3].bLongPressStart:= FALSE;
	arrButtons[3].bLongPressRepeat:= FALSE;	
	arrButtons[3].bLongPressStop:= FALSE;	
	arrButtons[3].bButtonFree := TRUE;
END_IF
END_ACTION

ACTION A_Sort_Event_Button4:

IF arrPushButtonEvent[4].1 THEN
	arrButtons[4].bPressed:= TRUE;
	arrButtons[4].bReleased:= FALSE;
END_IF

IF arrPushButtonEvent[4].0 THEN
	arrButtons[4].bPressed:= FALSE;
	arrButtons[4].bReleased:= TRUE;
END_IF

IF arrPushButtonEvent[4].2 THEN
	arrButtons[4].bShortPress:= TRUE;
END_IF

IF arrPushButtonEvent[4].3 THEN
	arrButtons[4].bDoublePress:= TRUE;
END_IF

IF arrPushButtonEvent[4].4 THEN
	arrButtons[4].bLongPressStop:= FALSE;
	arrButtons[4].bLongPressStart:= TRUE;
	arrButtons[4].bLongPressRepeat:= FALSE;	
END_IF

arrButtons[4].bLongPressRepeat:= arrPushButtonEvent[4].5 ;

IF arrPushButtonEvent[4].6 THEN
	arrButtons[4].bLongPressStop:= TRUE;
	arrButtons[4].bLongPressStart:= FALSE;
	arrButtons[4].bLongPressRepeat:= FALSE;	
END_IF

IF arrPushButtonEvent[4].7 THEN
	arrButtons[4].bPressed:= FALSE;
	arrButtons[4].bReleased:= FALSE;
	arrButtons[4].bShortPress:= FALSE;
	arrButtons[4].bDoublePress:= FALSE;	
	arrButtons[4].bLongPressStart:= FALSE;
	arrButtons[4].bLongPressRepeat:= FALSE;	
	arrButtons[4].bLongPressStop:= FALSE;	
	arrButtons[4].bButtonFree := TRUE;
END_IF
END_ACTION

ACTION A_Sort_Event_Button5:

IF arrPushButtonEvent[5].1 THEN
	arrButtons[5].bPressed:= TRUE;
	arrButtons[5].bReleased:= FALSE;
END_IF

IF arrPushButtonEvent[5].0 THEN
	arrButtons[5].bPressed:= FALSE;
	arrButtons[5].bReleased:= TRUE;
END_IF

IF arrPushButtonEvent[5].2 THEN
	arrButtons[5].bShortPress:= TRUE;
END_IF

IF arrPushButtonEvent[5].3 THEN
	arrButtons[5].bDoublePress:= TRUE;
END_IF

IF arrPushButtonEvent[5].4 THEN
	arrButtons[5].bLongPressStop:= FALSE;
	arrButtons[5].bLongPressStart:= TRUE;
	arrButtons[5].bLongPressRepeat:= FALSE;	
END_IF

arrButtons[5].bLongPressRepeat:= arrPushButtonEvent[5].5 ;

IF arrPushButtonEvent[5].6 THEN
	arrButtons[5].bLongPressStop:= TRUE;
	arrButtons[5].bLongPressStart:= FALSE;
	arrButtons[5].bLongPressRepeat:= FALSE;	
END_IF

IF arrPushButtonEvent[5].7 THEN
	arrButtons[5].bPressed:= FALSE;
	arrButtons[5].bReleased:= FALSE;
	arrButtons[5].bShortPress:= FALSE;
	arrButtons[5].bDoublePress:= FALSE;	
	arrButtons[5].bLongPressStart:= FALSE;
	arrButtons[5].bLongPressRepeat:= FALSE;	
	arrButtons[5].bLongPressStop:= FALSE;	
	arrButtons[5].bButtonFree := TRUE;
END_IF
END_ACTION

ACTION A_Sort_Event_Button6:

IF arrPushButtonEvent[6].1 THEN
	arrButtons[6].bPressed:= TRUE;
	arrButtons[6].bReleased:= FALSE;
END_IF

IF arrPushButtonEvent[6].0 THEN
	arrButtons[6].bPressed:= FALSE;
	arrButtons[6].bReleased:= TRUE;
END_IF

IF arrPushButtonEvent[6].2 THEN
	arrButtons[6].bShortPress:= TRUE;
END_IF

IF arrPushButtonEvent[6].3 THEN
	arrButtons[6].bDoublePress:= TRUE;
END_IF

IF arrPushButtonEvent[6].4 THEN
	arrButtons[6].bLongPressStop:= FALSE;
	arrButtons[6].bLongPressStart:= TRUE;
	arrButtons[6].bLongPressRepeat:= FALSE;	
END_IF

arrButtons[6].bLongPressRepeat:= arrPushButtonEvent[6].5 ;

IF arrPushButtonEvent[6].6 THEN
	arrButtons[6].bLongPressStop:= TRUE;
	arrButtons[6].bLongPressStart:= FALSE;
	arrButtons[6].bLongPressRepeat:= FALSE;	
END_IF

IF arrPushButtonEvent[6].7 THEN
	arrButtons[6].bPressed:= FALSE;
	arrButtons[6].bReleased:= FALSE;
	arrButtons[6].bShortPress:= FALSE;
	arrButtons[6].bDoublePress:= FALSE;	
	arrButtons[6].bLongPressStart:= FALSE;
	arrButtons[6].bLongPressRepeat:= FALSE;	
	arrButtons[6].bLongPressStop:= FALSE;	
	arrButtons[6].bButtonFree := TRUE;
END_IF
END_ACTION

ACTION A_Sort_Event_Button7:

IF arrPushButtonEvent[7].1 THEN
	arrButtons[7].bPressed:= TRUE;
	arrButtons[7].bReleased:= FALSE;
END_IF

IF arrPushButtonEvent[7].0 THEN
	arrButtons[7].bPressed:= FALSE;
	arrButtons[7].bReleased:= TRUE;
END_IF

IF arrPushButtonEvent[7].2 THEN
	arrButtons[7].bShortPress:= TRUE;
END_IF

IF arrPushButtonEvent[7].3 THEN
	arrButtons[7].bDoublePress:= TRUE;
END_IF

IF arrPushButtonEvent[7].4 THEN
	arrButtons[7].bLongPressStop:= FALSE;
	arrButtons[7].bLongPressStart:= TRUE;
	arrButtons[7].bLongPressRepeat:= FALSE;	
END_IF

arrButtons[7].bLongPressRepeat:= arrPushButtonEvent[7].5 ;

IF arrPushButtonEvent[7].6 THEN
	arrButtons[7].bLongPressStop:= TRUE;
	arrButtons[7].bLongPressStart:= FALSE;
	arrButtons[7].bLongPressRepeat:= FALSE;	
END_IF

IF arrPushButtonEvent[7].7 THEN
	arrButtons[7].bPressed:= FALSE;
	arrButtons[7].bReleased:= FALSE;
	arrButtons[7].bShortPress:= FALSE;
	arrButtons[7].bDoublePress:= FALSE;	
	arrButtons[7].bLongPressStart:= FALSE;
	arrButtons[7].bLongPressRepeat:= FALSE;	
	arrButtons[7].bLongPressStop:= FALSE;	
	arrButtons[7].bButtonFree := TRUE;
END_IF
END_ACTION

ACTION A_Sort_Event_Button8:

IF arrPushButtonEvent[8].1 THEN
	arrButtons[8].bPressed:= TRUE;
	arrButtons[8].bReleased:= FALSE;
END_IF

IF arrPushButtonEvent[8].0 THEN
	arrButtons[8].bPressed:= FALSE;
	arrButtons[8].bReleased:= TRUE;
END_IF

IF arrPushButtonEvent[8].2 THEN
	arrButtons[8].bShortPress:= TRUE;
END_IF

IF arrPushButtonEvent[8].3 THEN
	arrButtons[8].bDoublePress:= TRUE;
END_IF

IF arrPushButtonEvent[8].4 THEN
	arrButtons[8].bLongPressStop:= FALSE;
	arrButtons[8].bLongPressStart:= TRUE;
	arrButtons[8].bLongPressRepeat:= FALSE;	
END_IF

arrButtons[8].bLongPressRepeat:= arrPushButtonEvent[8].5 ;

IF arrPushButtonEvent[8].6 THEN
	arrButtons[8].bLongPressStop:= TRUE;
	arrButtons[8].bLongPressStart:= FALSE;
	arrButtons[8].bLongPressRepeat:= FALSE;	
END_IF

IF arrPushButtonEvent[8].7 THEN
	arrButtons[8].bPressed:= FALSE;
	arrButtons[8].bReleased:= FALSE;
	arrButtons[8].bShortPress:= FALSE;
	arrButtons[8].bDoublePress:= FALSE;	
	arrButtons[8].bLongPressStart:= FALSE;
	arrButtons[8].bLongPressRepeat:= FALSE;	
	arrButtons[8].bLongPressStop:= FALSE;	
	arrButtons[8].bButtonFree := TRUE;
END_IF
END_ACTION

END_FUNCTION_BLOCK

// POUs/DALI/DALI_Devices/Lunatone/FB_DALI_Lunatone_MC2_OLD
FUNCTION_BLOCK FB_DALI_Lunatone_MC2_OLD
VAR_INPUT
	byShrtAdr					: BYTE;
	bInitialize					: BOOL := TRUE;
	ipCommunication				: I_DALICommunication;
	DALI_LINE_NUM				: INT := 1;	
END_VAR
VAR_OUTPUT
	bInitErr: BOOL;
	bInitDone: BOOL;
	arrButtons					: ARRAY [1..10] OF BOOL;

END_VAR
VAR
	
	fbButton: FB_DALI_Lunatone_MC(0);
	_bEnablePushButton				:	BOOL := TRUE; // A TRUE at this input enables the instance for detecting movement. A FALSE at this input causes the sending of events from this instance to be disabled.
	_nEventFilterPushButton			:	BYTE := 2#1000_0011; // Setting of the eventfilter. If the respective bit is set, the corresponding event is active / Bit 0 : Button Released / Bit 1 : Button Pressed / Bit 2 : Short Press / Bit 3 : Double Press / Bit 4 : Long Press Start / Bit 5 : Long Press Repeat / Bit 6 : Long Press Stop / Bit 7 : Button Free / Button Stuck
	_nDoubleTimerPushButton			:	UINT := 0; // Time (0, tDoubleMin…2000 ms) to distinguish between a single and a double button press..
	_nRepeatTimerPushButton			:	UINT := 160; // Interval (100…2000 ms) of repetitive events in the case of a long button press.
	_nShortTimerPushButton			:	UINT := 500; // Time (tShortMin...5100 ms) to distinguish between a long and a short button press. tShortMin is a manufacturer-specific value.
	_nStuckTimerPushButton			:	BYTE := 20; // Time (5…255 s) after whose expiry the push button no longer represents a long button press. The push button is stuck.
	_eEventPriorityPushButton		:	E_DALIEventPriority := E_DALIEventPriority.Middle;  // Setting of the event priority (Low, MiddleLow, Middle, MiddleHigh).

	tDelayTime: TIME;
	fbDelaySetupDALIDevice: Ton;
	bInitSensor: BOOL;
	nPushButton1Event: WORD;
	nPushButton2Event: WORD;
	nPushButton3Event: WORD;
	nPushButton4Event: WORD;
	bPressed: BOOL;
	fbInitDone: F_TRIG;
	bInitializing: BOOL;
	bInitTimeOut: BOOL;
	fbInitTimeOut: TON;
END_VAR


fbButton.ipDALICommunication := ipCommunication;

IF ipCommunication <> 0 THEN
	A_LunatonButton();
END_IF

ACTION A_LunatonButton:

fbButton.bEnablePushButton1 := _bEnablePushButton;
fbButton.bEnablePushButton2 := _bEnablePushButton;
fbButton.bEnablePushButton3 := _bEnablePushButton;
fbButton.bEnablePushButton4 := _bEnablePushButton;

fbButton.eEventPriorityPushButton1 := _eEventPriorityPushButton;
fbButton.eEventPriorityPushButton2 := _eEventPriorityPushButton;
fbButton.eEventPriorityPushButton3 := _eEventPriorityPushButton;
fbButton.eEventPriorityPushButton4 := _eEventPriorityPushButton;

fbButton.nEventFilterPushButton1 := _nEventFilterPushButton; 
fbButton.nEventFilterPushButton2 := _nEventFilterPushButton; 
fbButton.nEventFilterPushButton3 := _nEventFilterPushButton; 
fbButton.nEventFilterPushButton4 := _nEventFilterPushButton; 


fbButton.nDoubleTimerPushButton1 := _nDoubleTimerPushButton;
fbButton.nDoubleTimerPushButton2 := _nDoubleTimerPushButton;
fbButton.nDoubleTimerPushButton3 := _nDoubleTimerPushButton;
fbButton.nDoubleTimerPushButton4 := _nDoubleTimerPushButton;

fbButton.nRepeatTimerPushButton1 := _nRepeatTimerPushButton;
fbButton.nRepeatTimerPushButton2 := _nRepeatTimerPushButton;
fbButton.nRepeatTimerPushButton3 := _nRepeatTimerPushButton;
fbButton.nRepeatTimerPushButton4 := _nRepeatTimerPushButton;

fbButton.nShortTimerPushButton1 := _nShortTimerPushButton;
fbButton.nShortTimerPushButton2 := _nShortTimerPushButton;
fbButton.nShortTimerPushButton3 := _nShortTimerPushButton;
fbButton.nShortTimerPushButton4 := _nShortTimerPushButton;

fbButton.nStuckTimerPushButton1 := _nStuckTimerPushButton;
fbButton.nStuckTimerPushButton2 := _nStuckTimerPushButton;
fbButton.nStuckTimerPushButton3 := _nStuckTimerPushButton;
fbButton.nStuckTimerPushButton4 := _nStuckTimerPushButton;

//Calculate delay time for init sensor
tDelayTime := INT_TO_TIME((BYTE_TO_INT(byShrtAdr) * 400));	
fbDelaySetupDALIDevice(IN:= bInitialize , PT:=tDelayTime , Q=> , ET=> );	
	
IF fbDelaySetupDALIDevice.q AND NOT GVL_DALI.arrbBlockDTR[DALI_LINE_NUM] AND NOT (bInitDone OR bInitErr) THEN
	bInitSensor:= TRUE;
	GVL_DALI.arrbBlockDTR[DALI_LINE_NUM]:= TRUE;
END_IF

fbButton(
	bInitialize:= bInitSensor , 
	nShortAddress:= byShrtAdr, 
	nOptions:= , 
	bQueryInputValue1:= , 
	bQueryInputValue2:= , 
	bQueryInputValue3:= , 
	bQueryInputValue4:= , 
	bInitializing=> bInitializing, 
	bReadingInputValue1=> , 
	bReadingInputValue2=> , 
	bReadingInputValue3=> , 
	bReadingInputValue4=> , 
	nPushButton1Event=> nPushButton1Event, 
	nPushButton2Event=> nPushButton2Event, 
	nPushButton3Event=> nPushButton3Event, 
	nPushButton4Event=> nPushButton4Event);


fbInitDone(CLK:=bInitializing );	
	IF fbInitDone.Q THEN
		IF NOT bInitTimeOut THEN
			bInitDone := TRUE;
			GVL_DALI.arrbBlockDTR[DALI_LINE_NUM]:= FALSE;
		ELSE
			bInitErr := TRUE;
			GVL_DALI.arrbBlockDTR[DALI_LINE_NUM]:= FALSE;
		END_IF
	END_IF
	
fbInitTimeOut(IN:=bInitSensor, PT:= T#10S); 
IF fbInitTimeOut.Q THEN
	bInitErr := TRUE;
	GVL_DALI.arrbBlockDTR[DALI_LINE_NUM]:= FALSE;
END_IF


IF nPushButton1Event.0 OR nPushButton1Event.7 THEN
	arrButtons[1] := FALSE;
END_IF
IF nPushButton1Event.1 THEN
	arrButtons[1] := TRUE;
END_IF

IF nPushButton2Event.0 OR nPushButton2Event.7THEN
	arrButtons[2] := FALSE;
END_IF
IF nPushButton2Event.1 THEN
	arrButtons[2] := TRUE;
END_IF

IF nPushButton3Event.0 OR nPushButton3Event.7THEN
	arrButtons[3] := FALSE;
END_IF
IF nPushButton3Event.1 THEN
	arrButtons[3] := TRUE;
END_IF

IF nPushButton4Event.0 OR nPushButton4Event.7THEN
	arrButtons[4] := FALSE;
END_IF
IF nPushButton4Event.1 THEN
	arrButtons[4] := TRUE;
END_IF
END_ACTION

END_FUNCTION_BLOCK

// POUs/DALI/DALI_Devices/Lunatone/FB_DALI_Lunatone_ROT
FUNCTION_BLOCK FB_DALI_Lunatone_ROT
VAR_INPUT
	byShrtAdr					: BYTE;
	bInitialize					: BOOL := TRUE;
	ipCommunication				: I_DALICommunication;
	DALI_LINE_NUM				: INT := 1;	
END_VAR
VAR_OUTPUT
	bInitErr: BOOL;
	bInitDone: BOOL;
	stRotation				: ST_ROT;

END_VAR
VAR
	
	fbRotation						: FB_DALI_Lunatone_ROT_D2I_Mode(0);
	_bEnablePushButton				:	BOOL := TRUE; // A TRUE at this input enables the instance for detecting movement. A FALSE at this input causes the sending of events from this instance to be disabled.
	_nEventFilterPushButton			:	BYTE := 2#1000_0011; // Setting of the eventfilter. If the respective bit is set, the corresponding event is active / Bit 0 : Button Released / Bit 1 : Button Pressed / Bit 2 : Short Press / Bit 3 : Double Press / Bit 4 : Long Press Start / Bit 5 : Long Press Repeat / Bit 6 : Long Press Stop / Bit 7 : Button Free / Button Stuck
	_nDoubleTimerPushButton			:	UINT := 0; // Time (0, tDoubleMin…2000 ms) to distinguish between a single and a double button press.
	_nRepeatTimerPushButton			:	UINT := 160; // Interval (100…2000 ms) of repetitive events in the case of a long button press.
	_nShortTimerPushButton			:	UINT := 500; // Time (tShortMin...5100 ms) to distinguish between a long and a short button press. tShortMin is a manufacturer-specific value.
	_nStuckTimerPushButton			:	BYTE := 20; // Time (5…255 s) after whose expiry the push button no longer represents a long button press. The push button is stuck.
	_eEventPriorityPushButton		:	E_DALIEventPriority := E_DALIEventPriority.Middle;  // Setting of the event priority (Low, MiddleLow, Middle, MiddleHigh).

	// Parameters Rotation
	_bEnableRotation				:	BOOL := TRUE; // A TRUE at this input enables the instance for measuring the brightness. A FALSE at this input causes the sending of events from this instance to be disabled.
	_nEventFilterRotation			:	BYTE := 2#0000_0111; // Setting of the eventfilter. If the respective bit is set, the corresponding event is active 
	_eEventPriorityRotation			:	E_DALIEventPriority := E_DALIEventPriority.MiddleLow; // Setting of the event priority (Low, MiddleLow, Middle, MiddleHigh).

	// Parameters POsition
	_bEnablePosition				:	BOOL := FALSE; // The instance can be enabled or disabled on the DALI control device. If this property is FALSE, sending events from this instance is disabled. However, the actual value of the instance can still be queried via the input bQueryInputValue.
	_nReportTimerPosition			:	BYTE := 0; // Time (0…255 s) after which the pending event of the measurement is repeated if no other event has occurred in the meantime.
	_nDeadtimeTimerPosition			:	UINT := 100; // Dead time (0...12750 ms) to ensure that not too many events are sent in succession. An event is only sent after expiry of the dead time timer. The dead time timer is restarted each time an event is sent.
	_eEventPriorityPosition			:	E_DALIEventPriority := E_DALIEventPriority.Middle; // Setting of the event priority (Low, MiddleLow, Middle, MiddleHigh).
	
	tDelayTime: TIME;
	fbDelaySetupDALIDevice: Ton;
	bInitSensor: BOOL;
	nPushButton1Event: WORD;
	nPushButton2Event: WORD;
	nPushButton3Event: WORD;
	nPushButton4Event: WORD;
	fbInitDone: F_TRIG;
	bInitializing: BOOL;
	bInitTimeOut: BOOL;
	fbInitTimeOut: TON;
	
	fbCheckButton_TON: TON;
	fbCheckRotation_TON: TON;
	
END_VAR

fbRotation.ipDALICommunication := ipCommunication;

IF ipCommunication <> 0 THEN
	A_LunatonRotation();
END_IF

ACTION A_LunatonRotation:
//Push function
fbRotation.bEnablePushButton 		:= _bEnablePushButton;
fbRotation.eEventPriorityButton 	:= _eEventPriorityPushButton;
fbRotation.nDoubleTimerPushButton 	:= _nDoubleTimerPushButton;
fbRotation.nEventFilterPushButton 	:= _nEventFilterPushButton; 
fbRotation.nRepeatTimerPushButton 	:= _nRepeatTimerPushButton;
fbRotation.nShortTimerPushButton 	:= _nShortTimerPushButton;
fbRotation.nStuckTimerPushButton 	:= _nStuckTimerPushButton;
//Rotation direction
fbRotation.bEnableRotation 			:= _bEnableRotation;
fbRotation.eEventPriorityRotation	:= _eEventPriorityRotation;
fbRotation.nEventFilterRotation 	:= _nEventFilterRotation;
//Position read out
fbRotation.bEnablePosition 			:= _bEnablePosition;
fbRotation.eEventPriorityPosition 	:= _eEventPriorityPosition;
fbRotation.nDeadtimerPosition 		:= _nDeadtimeTimerPosition;
fbRotation.nReportTimePosition 		:= _nReportTimerPosition; 


//Calculate delay time for init sensor
tDelayTime := INT_TO_TIME((BYTE_TO_INT(byShrtAdr) * 400));	
fbDelaySetupDALIDevice(IN:= bInitialize , PT:=tDelayTime , Q=> , ET=> );	
	
IF fbDelaySetupDALIDevice.q AND NOT GVL_DALI.arrbBlockDTR[DALI_LINE_NUM] AND NOT (bInitDone OR bInitErr) THEN
	bInitSensor:= TRUE;
	GVL_DALI.arrbBlockDTR[DALI_LINE_NUM]:= TRUE;
END_IF

fbRotation(
	bInitialize:= bInitialize, 
	nShortAddress:= byShrtAdr, 
	bQueryPushBotton:=fbCheckButton_TON.Q , 
	bQueryRotation:= fbCheckRotation_TON.Q, 
	bQueryPosition:= , 
	bBusy=> , 
	bError=> , 
	nErrorId=> , 
	bInitializing=> bInitializing, 
	bReadingPushbotton=> , 
	bReadingRotation=> , 
	bReadingPosition=> , 
	nPushBotton=> , 
	nRotation=> , 
	nPosition=> , 
	stROTdata=> stRotation , 
	bPressed=> , 
	bReleased=> , 
	bCW=> , 
	bCCW=> , 
	bNeutral=> );


fbInitDone(CLK:=bInitializing );	
	IF fbInitDone.Q THEN
		IF NOT bInitTimeOut THEN
			bInitDone := TRUE;
			GVL_DALI.arrbBlockDTR[DALI_LINE_NUM]:= FALSE;
		ELSE
			bInitErr := TRUE;
			GVL_DALI.arrbBlockDTR[DALI_LINE_NUM]:= FALSE;
		END_IF
	END_IF
	
fbInitTimeOut(IN:=bInitSensor, PT:= T#10S); 

IF fbInitTimeOut.Q THEN
	bInitErr := TRUE;
	GVL_DALI.arrbBlockDTR[DALI_LINE_NUM]:= FALSE;
END_IF


fbCheckButton_TON(IN:= stRotation.bPressed AND NOT fbCheckButton_TON.Q, PT:= T#2S , Q=> , ET=> );
fbCheckRotation_TON(IN:= (stRotation.bCCW OR stRotation.bCW) AND NOT fbCheckRotation_TON.Q , PT:= T#1S , Q=> , ET=> );
END_ACTION

END_FUNCTION_BLOCK

// POUs/DALI/Lunatone/FB_DALI_Lunatone_ROT_D2I_Mode
// This function block is an example of a DALI-2 input device.
FUNCTION_BLOCK PUBLIC FB_DALI_Lunatone_ROT_D2I_Mode
VAR_INPUT
	bInitialize						:	BOOL := FALSE; // The configuration of the DALI control device is started by a positive edge at this input.
	nShortAddress					:	BYTE := 0; // Short address of the DALI control device (0...63).
	bQueryPushBotton				:	BOOL := FALSE; // The Push botton is queried manually and event-independently by a rising edge at this input.
	bQueryRotation					:	BOOL := FALSE; // The rotation direction is queried manually and event-independently by a rising edge at this input.
	bQueryPosition					:	BOOL := FALSE; // The current position is queried manually and event-independently by a rising edge at this input.
END_VAR
VAR_OUTPUT
	bBusy							:	BOOL; // When the function block is activated the output is set, and it remains active until execution of the command has been completed.
	bError							:	BOOL; // This output is switched to TRUE if an error occurs during the execution of a command.
	nErrorId						:	UDINT; // Contains the error code of the most recently executed command. Error 1...1000 comes from the Tc3_DALI and error codes > 1000 are specific error codes of this FB.
	bInitializing					:	BOOL; // The output is set as soon as the initialization of the DALI control device has been started, and remains active until all DALI commands have been executed.
	bReadingPushbotton				:	BOOL; // The output is TRUE as long as values of the instance of the motion sensor are being read by the DALI control device.
	bReadingRotation				:	BOOL; // The output is TRUE as long as values of the instance of the Rotation direction are being read by the DALI control device.
	bReadingPosition				:	BOOL; // The output is TRUE as long as values of the instance of the position of the unit are being read by the DALI control device.
	nPushBotton						:	WORD; // The output outputs the events for the push button via one bit for one cycle.
	nRotation						:	WORD; // The output outputs the events for the push button via one bit for one cycle.
	nPosition						:	LWORD; // Outputs the measured value of the position measurement.
	stROTdata						: 	ST_ROT;
	bPressed						: 	BOOL;
	bReleased						: 	BOOL;
	bCW								: 	BOOL;
	bCCW							: 	BOOL;
	bNeutral						: 	BOOL;
END_VAR
VAR
	nStep							:	INT;
	rtrigInitialize					:	R_TRIG;
	rtrigReadingPushBotton			:	R_TRIG;
	rtrigReadingRotation			:	R_TRIG;
	rtrigReadingPosition			:	R_TRIG;
	tonDelay						:	TON;
	bParameterInvalid				:	BOOL := FALSE;
	bInitializePreset				:	BOOL := FALSE;
	bInit							:	BOOL;
	rtrigError103Generic			:	R_TRIG;
	ftrigError103Generic			:	F_TRIG;
	rtrigError301PushButton			:	R_TRIG;
	ftrigError301PushButton			:	F_TRIG;
	rtrigError301Rotation			:	R_TRIG;
	ftrigError301Rotation			:	F_TRIG;
	rtrigError302AbsoluteInputDevice:	R_TRIG;
	ftrigError302AbsoluteInputDevice:	F_TRIG;
	nShortAddressCheck				:	BYTE;

	{region 'Backing Variables'}
	_ipDALICommunication			:	I_DALICommunication;
	// Parameters Occupancy
	_bEnablePushButton				:	BOOL := TRUE; // A TRUE at this input enables the instance for detecting movement. A FALSE at this input causes the sending of events from this instance to be disabled.
	_nEventFilterPushButton			:	BYTE := 2#1000_0011; // Setting of the eventfilter. If the respective bit is set, the corresponding event is active / Bit 0 : Button Released / Bit 1 : Button Pressed / Bit 2 : Short Press / Bit 3 : Double Press / Bit 4 : Long Press Start / Bit 5 : Long Press Repeat / Bit 6 : Long Press Stop / Bit 7 : Button Free / Button Stuck
	_nDoubleTimerPushButton			:	UINT := 0; // Time (0, tDoubleMin…2000 ms) to distinguish between a single and a double button press..
	_nRepeatTimerPushButton			:	UINT := 160; // Interval (100…2000 ms) of repetitive events in the case of a long button press.
	_nShortTimerPushButton			:	UINT := 500; // Time (tShortMin...5100 ms) to distinguish between a long and a short button press. tShortMin is a manufacturer-specific value.
	_nStuckTimerPushButton			:	BYTE := 20; // Time (5…255 s) after whose expiry the push button no longer represents a long button press. The push button is stuck.
	_eEventPriorityPushButton		:	E_DALIEventPriority := E_DALIEventPriority.Middle;  // Setting of the event priority (Low, MiddleLow, Middle, MiddleHigh).

	// Parameters Rotation
	_bEnableRotation				:	BOOL := TRUE; // A TRUE at this input enables the instance for measuring the brightness. A FALSE at this input causes the sending of events from this instance to be disabled.
	_nEventFilterRotation			:	BYTE := 2#0000_0111; // Setting of the eventfilter. If the respective bit is set, the corresponding event is active 
	_eEventPriorityRotation			:	E_DALIEventPriority := E_DALIEventPriority.MiddleLow; // Setting of the event priority (Low, MiddleLow, Middle, MiddleHigh).

	// Parameters Rotation
	_bEnablePosition				:	BOOL := FALSE; // The instance can be enabled or disabled on the DALI control device. If this property is FALSE, sending events from this instance is disabled. However, the actual value of the instance can still be queried via the input bQueryInputValue.
	_nReportTimerPosition			:	BYTE := 0; // Time (0…255 s) after which the pending event of the measurement is repeated if no other event has occurred in the meantime.
	_nDeadtimeTimerPosition			:	UINT := 100; // Dead time (0...12750 ms) to ensure that not too many events are sent in succession. An event is only sent after expiry of the dead time timer. The dead time timer is restarted each time an event is sent.
	_eEventPriorityPosition			:	E_DALIEventPriority := E_DALIEventPriority.Middle; // Setting of the event priority (Low, MiddleLow, Middle, MiddleHigh).
	{endregion}

	{region 'Function Blocks for the DALI commands'}
	fb103ControlDevice				:	FB_DALI103ControlDevice(0);
	fb301PushButton					:	FB_DALI301PushButton(0);
	fb301Rotation					:	FB_DALI301PushButton(0);
	fb302AbsoluteInputDevice		:	FB_DALI302AbsoluteInputDevice(0);
		 
	fbSavePersistentVariables		:	FB_DALI103SavePersistentVariables(0);
	fbStartQuiescentMode			:	FB_DALI103StartQuiescentMode(0);
	fbStopQuiescentMode				:	FB_DALI103StopQuiescentMode(0);
	{endregion}
END_VAR

IF (NOT bInit) THEN
	bInit := TRUE;
	THIS^.SetCommunication();
	nErrorId := THIS^.CheckParameters();
	bError := (nErrorId > 0);
	nStep := 0;
END_IF

rtrigInitialize(CLK := bInitialize);
IF (rtrigInitialize.Q AND NOT bInitializing) THEN
	bInitializePreset := TRUE;
END_IF
IF (bInitializePreset AND NOT bReadingPushbotton AND NOT bReadingRotation AND NOT bReadingPosition) THEN
	bInitializePreset := FALSE;
	bInitializing := TRUE;
	THIS^.SetCommunication();
	nErrorId := THIS^.CheckParameters();
	bError := (nErrorId > 0);
	IF (NOT bError) THEN
		nStep := 10; // Initialize
	ELSE
		nPushBotton := 1;
		nRotation := 4;
		nPosition := 0;
		nStep := 0;
	END_IF
END_IF

CASE nStep OF
0:
	bInitializing := FALSE;

{region 'Initialize Control Device'}
10: // Device
	fb103ControlDevice.bEnableApplicationController := TRUE;
	fb103ControlDevice.bEnablePowerCycleNotification := FALSE;
	fb103ControlDevice.nOperatingMode := 164;
	fb103ControlDevice(	bInitialize := TRUE,
						bGetPowerCycleNotifications := FALSE,
						nShortAddress := nShortAddress);
	IF (NOT fb103ControlDevice.bInitializing) THEN
		IF (NOT fb103ControlDevice.bError) THEN
			nStep := 20;
		ELSE
			nErrorId := fb103ControlDevice.ipResultMessage.nEventId;
			bError := TRUE;
			bInitializing := FALSE;
			nPushBotton := 1;
			nRotation := 4;
			nPosition := 0;
			nStep := 0;
		END_IF
		fb103ControlDevice(bInitialize := FALSE);
	END_IF

20: // Start Quiescent Mode
	fbStartQuiescentMode(	bStart := TRUE,
							nAddress := nShortAddress,
							eAddressType := E_DALIAddressType.Short,
							eCommandPriority := E_DALICommandPriority.MiddleHigh);
	IF (NOT fbStartQuiescentMode.bBusy) THEN 
		IF (NOT fbStartQuiescentMode.bError) THEN
			nStep := 100;
		ELSE
			nErrorId := fbStartQuiescentMode.ipResultMessage.nEventId;
			bError := TRUE;
			bInitializing := FALSE;
			nPushBotton := 1;
			nRotation := 4;
			nPosition := 0;
			nStep := 0;
		END_IF
		fbStartQuiescentMode(bStart := FALSE);
	END_IF

100: // Instance 0 - Push botton
	fb301PushButton.bEnableInstance := _bEnablePushButton;
	fb301PushButton.nEventFilter := _nEventFilterPushButton;
	fb301PushButton.eEventPriority := _eEventPriorityPushButton;
	fb301PushButton.nDoubleTimer := _nDoubleTimerPushButton;
	fb301PushButton.nRepeatTimer := _nRepeatTimerPushButton;
	fb301PushButton.nShortTimer := _nShortTimerPushButton;
	fb301PushButton.nStuckTimer := _nStuckTimerPushButton;
		 
	fb301PushButton(	bInitialize := TRUE,
							bQueryInputValue := FALSE,
							bGetInputNotifications := FALSE,
							nShortAddress := nShortAddress,
							nInstanceNumber := 0);
	IF (NOT fb301PushButton.bInitializing) THEN
		IF (NOT fb301PushButton.bError) THEN
			nStep := 200;
		ELSE 
			nErrorId := fb301PushButton.ipResultMessage.nEventId;
			bError := TRUE;
			bInitializing := FALSE;
			nPushBotton := 1;
			nRotation := 4;
			nPosition := 0;
			nStep := 0;
		END_IF
		fb301PushButton(bInitialize := FALSE);
	END_IF

200: // Instance 1 - Rotation direction
	fb301Rotation.bEnableInstance := _bEnableRotation;
	fb301Rotation.eEventPriority := _eEventPriorityRotation;
	fb301Rotation.nEventFilter := _nEventFilterRotation;
	
	fb301Rotation(
		bInitialize:= TRUE, 
		nShortAddress:= nShortAddress, 
		nInstanceNumber:= 1, 
		bQueryInputValue:= FALSE, 
		bGetInputNotifications:= FALSE);	 

	IF (NOT fb301Rotation.bInitializing) THEN
		IF (NOT fb301Rotation.bError) THEN
			nStep := 300;
		ELSE 
			nErrorId := fb301Rotation.ipResultMessage.nEventId;
			bError := TRUE;
			bInitializing := FALSE;
			nPushBotton := 1;
			nRotation := 4;
			nPosition := 0;
			nStep := 0;
		END_IF
		fb301Rotation(bInitialize := FALSE);
	END_IF
		 
300: // Instance 3 - Position
	fb302AbsoluteInputDevice.bEnableInstance := _bEnablePosition;
	fb302AbsoluteInputDevice.eEventPriority := _eEventPriorityPosition;
	fb302AbsoluteInputDevice.nReportTimer := _nReportTimerPosition;
	fb302AbsoluteInputDevice.nDeadtimeTimer:= _nDeadtimeTimerPosition;	 
	fb302AbsoluteInputDevice(bInitialize:= TRUE, 
		nShortAddress:= nShortAddress, 
		nInstanceNumber:= 2, 
		nResolution:= 8, 
		bQueryInputValue:= FALSE);

	IF (NOT fb302AbsoluteInputDevice.bInitializing) THEN
		IF (NOT fb302AbsoluteInputDevice.bError) THEN
			nStep := 900;
		ELSE 
			nErrorId := fb302AbsoluteInputDevice.ipResultMessage.nEventId;
			bError := TRUE;
			bInitializing := FALSE;
			nPushBotton := 1;
			nRotation := 4;
			nPosition := 0;
		END_IF
		fb302AbsoluteInputDevice(bInitialize := FALSE);
	END_IF			  

	 
900: // Save Persistent Variables
	fbSavePersistentVariables(	bStart := TRUE,
								nAddress := nShortAddress,
								eAddressType := E_DALIAddressType.Short,
								eCommandPriority := E_DALICommandPriority.MiddleHigh);
	IF (NOT fbSavePersistentVariables.bBusy) THEN
		IF (NOT fbSavePersistentVariables.bError) THEN
			nStep := 910;
		ELSE
			nErrorId := fbSavePersistentVariables.ipResultMessage.nEventId;
			bError := TRUE;
			bInitializing := FALSE;
			nPushBotton := 1;
			nRotation := 4;
			nPosition := 0;
			nStep := 0;
		END_IF
		fbSavePersistentVariables(bStart := FALSE);
	END_IF

910: // Stop Quiescent Mode
	fbStopQuiescentMode(	bStart := TRUE,
							nAddress := nShortAddress,
							eAddressType := E_DALIAddressType.Short,
							eCommandPriority := E_DALICommandPriority.MiddleHigh);
	IF (NOT fbStopQuiescentMode.bBusy) THEN
		IF (NOT fbStopQuiescentMode.bError) THEN
			nStep := 920;
		ELSE
			nErrorId := fbStopQuiescentMode.ipResultMessage.nEventId;
			bError := TRUE;
			bInitializing := FALSE;
			nPushBotton := 1;
			nRotation := 4;
			nPosition := 0;
			nStep := 0;
		END_IF
		fbStopQuiescentMode(bStart := FALSE);
	END_IF

920: // Wait 1 sec. Device is saving the variables during this time.
	tonDelay(IN := TRUE, PT := T#1S);
	IF (tonDelay.Q) THEN
		tonDelay(IN := FALSE);
		nStep := 930;
	END_IF

